FUNCTION_BLOCK "HF3_IMCC_DT_FB2711"	// FB 2711
VERSION : 0.1
VAR
  PT_DT : TIME  := T#45S;
  K4_DTS_A1 : FB 2712;
  K4_DTS_A2 : FB 2712;
  K4_DTS_A3 : FB 2712;
  DTS_A1 : FB 2712;
  DTS_A2 : FB 2712;
  DTS_A4 : FB 2712;
  DTS_A6 : FB 2712;
  UOF_DT_A1 : FB 2712;
  UOF_DT_A2 : FB 2712;
  UOF_DT_A3 : FB 2712;
  UOF_DT_A4 : FB 2712;
  DTS_A5 : FB 2712;
  DTS_A3 : FB 2712;
END_VAR
BEGIN
NETWORK
TITLE =  K4-DTS-A1
      A     "IMCC_LOCK".K4_XK_A1_Stop;
      =     L 0.0;
      BLD   103;
      BLD   14;
      =     L 7.0;
      L     DINO;
      T     LW 5;
      CDB;
      OPN   DI [LW 5];
      TAR2  LD 1;
      OPN   DI 2291;
      L     DIW 604;
      OPN   DI [LW 5];
      T     #K4_DTS_A1.IN_RD;
      OPN   DI 6040;
      L     DIW 152;
      OPN   DI [LW 5];
      T     #K4_DTS_A1.SCtrl;
      OPN   DI 7005;
      L     DIW 312;
      OPN   DI [LW 5];
      T     #K4_DTS_A1.H_P_ALL_Ctrl;
      A     L 0.0;
      =     #K4_DTS_A1.Stop;
      BLD   11;
      L     W#16#1002;
      T     LW 10;
      L     2;
      T     LW 12;
      L     7004;
      T     LW 14;
      L     P#DBX 58.0;
      T     LD 16;
      L     W#16#1002;
      T     LW 20;
      L     2;
      T     LW 22;
      L     DINO;
      T     LW 24;
      +AR2  P#12.0;
      TAR2;
      LAR2  LD 1;
      T     LD 26;
      UC    "BLKMOV";
      {     P#L 10.0, P#L 8.0, P#L 20.0 };
      BLD   11;
      L     W#16#1002;
      T     LW 10;
      L     2;
      T     LW 12;
      L     7005;
      T     LW 14;
      L     P#DBX 4.0;
      T     LD 16;
      L     W#16#1002;
      T     LW 20;
      L     2;
      T     LW 22;
      L     DINO;
      T     LW 24;
      +AR2  P#14.0;
      TAR2;
      LAR2  LD 1;
      T     LD 26;
      UC    "BLKMOV";
      {     P#L 10.0, P#L 8.0, P#L 20.0 };
      BLD   11;
      L     W#16#1002;
      T     LW 10;
      L     2;
      T     LW 12;
      L     7005;
      T     LW 14;
      L     P#DBX 34.0;
      T     LD 16;
      L     W#16#1002;
      T     LW 20;
      L     2;
      T     LW 22;
      L     DINO;
      T     LW 24;
      +AR2  P#16.0;
      TAR2;
      LAR2  LD 1;
      T     LD 26;
      UC    "BLKMOV";
      {     P#L 10.0, P#L 8.0, P#L 20.0 };
      L     DBD [AR2,P#0.0];
      T     #K4_DTS_A1.PT;
      +AR2  P#4.0;
      UC    "HF3_IMCC_DT_FB2712";
      LAR2  LD 1;
      L     #K4_DTS_A1.qnWR;
      OPN   DI 2292;
      T     DIW 124;
      OPN   DI [LW 5];
      L     #K4_DTS_A1.TOHMI;
      OPN   DI 6004;
      T     DIW 482;
      OPN   DI [LW 5];
      A     #K4_DTS_A1.Refuse;
      OPN   DI 7006;
      =     DIX 5.0;
      OPN   DI [LW 5];
      A     #K4_DTS_A1.Open;
      OPN   DI 2555;
      =     DIX 3.1;
      OPN   DI [LW 5];
      CDB;
      BLD   15;
      NOP   0;
NETWORK
TITLE =  K4-DTS-A2
      A     "IMCC_LOCK".K4_DT_A2_Open;
      =     L 0.0;
      BLD   103;
      BLD   14;
      =     L 7.0;
      L     DINO;
      T     LW 5;
      CDB;
      OPN   DI [LW 5];
      TAR2  LD 1;
      OPN   DI 2291;
      L     DIW 606;
      OPN   DI [LW 5];
      T     DIW [AR2,P#110.0];
      OPN   DI 6040;
      L     DIW 154;
      OPN   DI [LW 5];
      T     DIW [AR2,P#112.0];
      OPN   DI 7005;
      L     DIW 312;
      OPN   DI [LW 5];
      T     DIW [AR2,P#114.0];
      A     L 0.0;
      =     DIX [AR2,P#116.0];
      BLD   11;
      L     W#16#1002;
      T     LW 10;
      L     2;
      T     LW 12;
      L     7004;
      T     LW 14;
      L     P#DBX 60.0;
      T     LD 16;
      L     W#16#1002;
      T     LW 20;
      L     2;
      T     LW 22;
      L     DINO;
      T     LW 24;
      +AR2  P#118.0;
      TAR2;
      LAR2  LD 1;
      T     LD 26;
      UC    "BLKMOV";
      {     P#L 10.0, P#L 8.0, P#L 20.0 };
      BLD   11;
      L     W#16#1002;
      T     LW 10;
      L     2;
      T     LW 12;
      L     7005;
      T     LW 14;
      L     P#DBX 4.0;
      T     LD 16;
      L     W#16#1002;
      T     LW 20;
      L     2;
      T     LW 22;
      L     DINO;
      T     LW 24;
      +AR2  P#120.0;
      TAR2;
      LAR2  LD 1;
      T     LD 26;
      UC    "BLKMOV";
      {     P#L 10.0, P#L 8.0, P#L 20.0 };
      BLD   11;
      L     W#16#1002;
      T     LW 10;
      L     2;
      T     LW 12;
      L     7005;
      T     LW 14;
      L     P#DBX 34.0;
      T     LD 16;
      L     W#16#1002;
      T     LW 20;
      L     2;
      T     LW 22;
      L     DINO;
      T     LW 24;
      +AR2  P#122.0;
      TAR2;
      LAR2  LD 1;
      T     LD 26;
      UC    "BLKMOV";
      {     P#L 10.0, P#L 8.0, P#L 20.0 };
      L     DBD [AR2,P#0.0];
      T     DID [AR2,P#124.0];
      +AR2  P#110.0;
      UC    "HF3_IMCC_DT_FB2712";
      LAR2  LD 1;
      L     DIW [AR2,P#128.0];
      OPN   DI 2292;
      T     DIW 126;
      OPN   DI [LW 5];
      L     DIW [AR2,P#130.0];
      OPN   DI 6004;
      T     DIW 484;
      OPN   DI [LW 5];
      A     DIX [AR2,P#132.0];
      OPN   DI 7006;
      =     DIX 5.1;
      OPN   DI [LW 5];
      A     DIX [AR2,P#132.1];
      OPN   DI 2555;
      =     DIX 3.2;
      OPN   DI [LW 5];
      CDB;
      BLD   15;
      NOP   0;
NETWORK
TITLE =  K4-DTS-A3
      A(;
      O     "IMCC_LOCK".K4_HPF_A1_Stop;
      O     "IMCC_LOCK".K4_XK_A1_Stop;
      );
      =     L 0.0;
      BLD   103;
      BLD   14;
      =     L 7.0;
      L     DINO;
      T     LW 5;
      CDB;
      OPN   DI [LW 5];
      TAR2  LD 1;
      OPN   DI 2291;
      L     DIW 608;
      OPN   DI [LW 5];
      T     DIW [AR2,P#216.0];
      OPN   DI 6040;
      L     DIW 156;
      OPN   DI [LW 5];
      T     DIW [AR2,P#218.0];
      OPN   DI 7005;
      L     DIW 312;
      OPN   DI [LW 5];
      T     DIW [AR2,P#220.0];
      A     L 0.0;
      =     DIX [AR2,P#222.0];
      BLD   11;
      L     W#16#1002;
      T     LW 10;
      L     2;
      T     LW 12;
      L     7004;
      T     LW 14;
      L     P#DBX 62.0;
      T     LD 16;
      L     W#16#1002;
      T     LW 20;
      L     2;
      T     LW 22;
      L     DINO;
      T     LW 24;
      +AR2  P#224.0;
      TAR2;
      LAR2  LD 1;
      T     LD 26;
      UC    "BLKMOV";
      {     P#L 10.0, P#L 8.0, P#L 20.0 };
      BLD   11;
      L     W#16#1002;
      T     LW 10;
      L     2;
      T     LW 12;
      L     7005;
      T     LW 14;
      L     P#DBX 4.0;
      T     LD 16;
      L     W#16#1002;
      T     LW 20;
      L     2;
      T     LW 22;
      L     DINO;
      T     LW 24;
      +AR2  P#226.0;
      TAR2;
      LAR2  LD 1;
      T     LD 26;
      UC    "BLKMOV";
      {     P#L 10.0, P#L 8.0, P#L 20.0 };
      BLD   11;
      L     W#16#1002;
      T     LW 10;
      L     2;
      T     LW 12;
      L     7005;
      T     LW 14;
      L     P#DBX 34.0;
      T     LD 16;
      L     W#16#1002;
      T     LW 20;
      L     2;
      T     LW 22;
      L     DINO;
      T     LW 24;
      +AR2  P#228.0;
      TAR2;
      LAR2  LD 1;
      T     LD 26;
      UC    "BLKMOV";
      {     P#L 10.0, P#L 8.0, P#L 20.0 };
      L     DBD [AR2,P#0.0];
      T     DID [AR2,P#230.0];
      +AR2  P#216.0;
      UC    "HF3_IMCC_DT_FB2712";
      LAR2  LD 1;
      L     DIW [AR2,P#234.0];
      OPN   DI 2292;
      T     DIW 128;
      OPN   DI [LW 5];
      L     DIW [AR2,P#236.0];
      OPN   DI 6004;
      T     DIW 486;
      OPN   DI [LW 5];
      A     DIX [AR2,P#238.0];
      OPN   DI 7006;
      =     DIX 5.2;
      OPN   DI [LW 5];
      A     DIX [AR2,P#238.1];
      OPN   DI 2555;
      =     DIX 3.3;
      OPN   DI [LW 5];
      CDB;
      BLD   15;
      NOP   0;
NETWORK
TITLE = DTS-A1
      A     "Always1";
      =     L 0.0;
      BLD   103;
      BLD   14;
      =     L 7.0;
      L     DINO;
      T     LW 5;
      CDB;
      OPN   DI [LW 5];
      TAR2  LD 1;
      OPN   DI 2291;
      L     DIW 676;
      OPN   DI [LW 5];
      T     DIW [AR2,P#322.0];
      OPN   DI 6040;
      L     DIW 60;
      OPN   DI [LW 5];
      T     DIW [AR2,P#324.0];
      OPN   DI 7005;
      L     DIW 312;
      OPN   DI [LW 5];
      T     DIW [AR2,P#326.0];
      A     L 0.0;
      =     DIX [AR2,P#328.0];
      BLD   11;
      L     W#16#1002;
      T     LW 10;
      L     2;
      T     LW 12;
      L     7004;
      T     LW 14;
      L     P#DBX 4.0;
      T     LD 16;
      L     W#16#1002;
      T     LW 20;
      L     2;
      T     LW 22;
      L     DINO;
      T     LW 24;
      +AR2  P#330.0;
      TAR2;
      LAR2  LD 1;
      T     LD 26;
      UC    "BLKMOV";
      {     P#L 10.0, P#L 8.0, P#L 20.0 };
      BLD   11;
      L     W#16#1002;
      T     LW 10;
      L     2;
      T     LW 12;
      L     7005;
      T     LW 14;
      L     P#DBX 0.0;
      T     LD 16;
      L     W#16#1002;
      T     LW 20;
      L     2;
      T     LW 22;
      L     DINO;
      T     LW 24;
      +AR2  P#332.0;
      TAR2;
      LAR2  LD 1;
      T     LD 26;
      UC    "BLKMOV";
      {     P#L 10.0, P#L 8.0, P#L 20.0 };
      BLD   11;
      L     W#16#1002;
      T     LW 10;
      L     2;
      T     LW 12;
      L     7005;
      T     LW 14;
      L     P#DBX 30.0;
      T     LD 16;
      L     W#16#1002;
      T     LW 20;
      L     2;
      T     LW 22;
      L     DINO;
      T     LW 24;
      +AR2  P#334.0;
      TAR2;
      LAR2  LD 1;
      T     LD 26;
      UC    "BLKMOV";
      {     P#L 10.0, P#L 8.0, P#L 20.0 };
      L     DBD [AR2,P#0.0];
      T     DID [AR2,P#336.0];
      +AR2  P#322.0;
      UC    "HF3_IMCC_DT_FB2712";
      LAR2  LD 1;
      L     DIW [AR2,P#340.0];
      OPN   DI 2292;
      T     DIW 196;
      OPN   DI [LW 5];
      L     DIW [AR2,P#342.0];
      OPN   DI 6004;
      T     DIW 518;
      OPN   DI [LW 5];
      A     DIX [AR2,P#344.0];
      OPN   DI 7006;
      =     DIX 2.0;
      OPN   DI [LW 5];
      A     DIX [AR2,P#344.1];
      OPN   DI 2555;
      =     DIX 0.2;
      OPN   DI [LW 5];
      CDB;
      BLD   15;
      NOP   0;
NETWORK
TITLE = DTS-A2
      A     "Always1";
      =     L 0.0;
      BLD   103;
      BLD   14;
      =     L 7.0;
      L     DINO;
      T     LW 5;
      CDB;
      OPN   DI [LW 5];
      TAR2  LD 1;
      OPN   DI 2291;
      L     DIW 678;
      OPN   DI [LW 5];
      T     DIW [AR2,P#428.0];
      OPN   DI 6040;
      L     DIW 62;
      OPN   DI [LW 5];
      T     DIW [AR2,P#430.0];
      OPN   DI 7005;
      L     DIW 312;
      OPN   DI [LW 5];
      T     DIW [AR2,P#432.0];
      A     L 0.0;
      =     DIX [AR2,P#434.0];
      BLD   11;
      L     W#16#1002;
      T     LW 10;
      L     2;
      T     LW 12;
      L     7004;
      T     LW 14;
      L     P#DBX 6.0;
      T     LD 16;
      L     W#16#1002;
      T     LW 20;
      L     2;
      T     LW 22;
      L     DINO;
      T     LW 24;
      +AR2  P#436.0;
      TAR2;
      LAR2  LD 1;
      T     LD 26;
      UC    "BLKMOV";
      {     P#L 10.0, P#L 8.0, P#L 20.0 };
      BLD   11;
      L     W#16#1002;
      T     LW 10;
      L     2;
      T     LW 12;
      L     7005;
      T     LW 14;
      L     P#DBX 0.0;
      T     LD 16;
      L     W#16#1002;
      T     LW 20;
      L     2;
      T     LW 22;
      L     DINO;
      T     LW 24;
      +AR2  P#438.0;
      TAR2;
      LAR2  LD 1;
      T     LD 26;
      UC    "BLKMOV";
      {     P#L 10.0, P#L 8.0, P#L 20.0 };
      BLD   11;
      L     W#16#1002;
      T     LW 10;
      L     2;
      T     LW 12;
      L     7005;
      T     LW 14;
      L     P#DBX 30.0;
      T     LD 16;
      L     W#16#1002;
      T     LW 20;
      L     2;
      T     LW 22;
      L     DINO;
      T     LW 24;
      +AR2  P#440.0;
      TAR2;
      LAR2  LD 1;
      T     LD 26;
      UC    "BLKMOV";
      {     P#L 10.0, P#L 8.0, P#L 20.0 };
      L     DBD [AR2,P#0.0];
      T     DID [AR2,P#442.0];
      +AR2  P#428.0;
      UC    "HF3_IMCC_DT_FB2712";
      LAR2  LD 1;
      L     DIW [AR2,P#446.0];
      OPN   DI 2292;
      T     DIW 198;
      OPN   DI [LW 5];
      L     DIW [AR2,P#448.0];
      OPN   DI 6004;
      T     DIW 520;
      OPN   DI [LW 5];
      A     DIX [AR2,P#450.0];
      OPN   DI 7006;
      =     DIX 2.1;
      OPN   DI [LW 5];
      A     DIX [AR2,P#450.1];
      OPN   DI 2555;
      =     DIX 0.3;
      OPN   DI [LW 5];
      CDB;
      BLD   15;
      NOP   0;
NETWORK
TITLE = DTS-A3
      A     "Always1";
      =     L 0.0;
      BLD   103;
      BLD   14;
      =     L 7.0;
      L     DINO;
      T     LW 5;
      CDB;
      OPN   DI [LW 5];
      TAR2  LD 1;
      OPN   DI 2291;
      L     DIW 680;
      OPN   DI [LW 5];
      T     DIW [AR2,P#1276.0];
      OPN   DI 6040;
      L     DIW 64;
      OPN   DI [LW 5];
      T     DIW [AR2,P#1278.0];
      OPN   DI 7005;
      L     DIW 312;
      OPN   DI [LW 5];
      T     DIW [AR2,P#1280.0];
      A     L 0.0;
      =     DIX [AR2,P#1282.0];
      BLD   11;
      L     W#16#1002;
      T     LW 10;
      L     2;
      T     LW 12;
      L     7004;
      T     LW 14;
      L     P#DBX 8.0;
      T     LD 16;
      L     W#16#1002;
      T     LW 20;
      L     2;
      T     LW 22;
      L     DINO;
      T     LW 24;
      +AR2  P#1284.0;
      TAR2;
      LAR2  LD 1;
      T     LD 26;
      UC    "BLKMOV";
      {     P#L 10.0, P#L 8.0, P#L 20.0 };
      BLD   11;
      L     W#16#1002;
      T     LW 10;
      L     2;
      T     LW 12;
      L     7005;
      T     LW 14;
      L     P#DBX 0.0;
      T     LD 16;
      L     W#16#1002;
      T     LW 20;
      L     2;
      T     LW 22;
      L     DINO;
      T     LW 24;
      +AR2  P#1286.0;
      TAR2;
      LAR2  LD 1;
      T     LD 26;
      UC    "BLKMOV";
      {     P#L 10.0, P#L 8.0, P#L 20.0 };
      BLD   11;
      L     W#16#1002;
      T     LW 10;
      L     2;
      T     LW 12;
      L     7005;
      T     LW 14;
      L     P#DBX 30.0;
      T     LD 16;
      L     W#16#1002;
      T     LW 20;
      L     2;
      T     LW 22;
      L     DINO;
      T     LW 24;
      +AR2  P#1288.0;
      TAR2;
      LAR2  LD 1;
      T     LD 26;
      UC    "BLKMOV";
      {     P#L 10.0, P#L 8.0, P#L 20.0 };
      L     DBD [AR2,P#0.0];
      T     DID [AR2,P#1290.0];
      +AR2  P#1276.0;
      UC    "HF3_IMCC_DT_FB2712";
      LAR2  LD 1;
      L     DIW [AR2,P#1294.0];
      OPN   DI 2292;
      T     DIW 200;
      OPN   DI [LW 5];
      L     DIW [AR2,P#1296.0];
      OPN   DI 6004;
      T     DIW 522;
      OPN   DI [LW 5];
      A     DIX [AR2,P#1298.0];
      OPN   DI 7006;
      =     DIX 2.2;
      OPN   DI [LW 5];
      A     DIX [AR2,P#1298.1];
      OPN   DI 2555;
      =     DIX 0.4;
      OPN   DI [LW 5];
      CDB;
      BLD   15;
      NOP   0;
NETWORK
TITLE = DTS-A4
      A     "Always1";
      =     L 0.0;
      BLD   103;
      BLD   14;
      =     L 7.0;
      L     DINO;
      T     LW 5;
      CDB;
      OPN   DI [LW 5];
      TAR2  LD 1;
      OPN   DI 2291;
      L     DIW 682;
      OPN   DI [LW 5];
      T     DIW [AR2,P#534.0];
      OPN   DI 6040;
      L     DIW 66;
      OPN   DI [LW 5];
      T     DIW [AR2,P#536.0];
      OPN   DI 7005;
      L     DIW 312;
      OPN   DI [LW 5];
      T     DIW [AR2,P#538.0];
      A     L 0.0;
      =     DIX [AR2,P#540.0];
      BLD   11;
      L     W#16#1002;
      T     LW 10;
      L     2;
      T     LW 12;
      L     7004;
      T     LW 14;
      L     P#DBX 10.0;
      T     LD 16;
      L     W#16#1002;
      T     LW 20;
      L     2;
      T     LW 22;
      L     DINO;
      T     LW 24;
      +AR2  P#542.0;
      TAR2;
      LAR2  LD 1;
      T     LD 26;
      UC    "BLKMOV";
      {     P#L 10.0, P#L 8.0, P#L 20.0 };
      BLD   11;
      L     W#16#1002;
      T     LW 10;
      L     2;
      T     LW 12;
      L     7005;
      T     LW 14;
      L     P#DBX 0.0;
      T     LD 16;
      L     W#16#1002;
      T     LW 20;
      L     2;
      T     LW 22;
      L     DINO;
      T     LW 24;
      +AR2  P#544.0;
      TAR2;
      LAR2  LD 1;
      T     LD 26;
      UC    "BLKMOV";
      {     P#L 10.0, P#L 8.0, P#L 20.0 };
      BLD   11;
      L     W#16#1002;
      T     LW 10;
      L     2;
      T     LW 12;
      L     7005;
      T     LW 14;
      L     P#DBX 30.0;
      T     LD 16;
      L     W#16#1002;
      T     LW 20;
      L     2;
      T     LW 22;
      L     DINO;
      T     LW 24;
      +AR2  P#546.0;
      TAR2;
      LAR2  LD 1;
      T     LD 26;
      UC    "BLKMOV";
      {     P#L 10.0, P#L 8.0, P#L 20.0 };
      L     DBD [AR2,P#0.0];
      T     DID [AR2,P#548.0];
      +AR2  P#534.0;
      UC    "HF3_IMCC_DT_FB2712";
      LAR2  LD 1;
      L     DIW [AR2,P#552.0];
      OPN   DI 2292;
      T     DIW 202;
      OPN   DI [LW 5];
      L     DIW [AR2,P#554.0];
      OPN   DI 6004;
      T     DIW 524;
      OPN   DI [LW 5];
      A     DIX [AR2,P#556.0];
      OPN   DI 7006;
      =     DIX 2.3;
      OPN   DI [LW 5];
      A     DIX [AR2,P#556.1];
      OPN   DI 2555;
      =     DIX 0.5;
      OPN   DI [LW 5];
      CDB;
      BLD   15;
      NOP   0;
NETWORK
TITLE = DTS-A5
      A     "Always1";
      =     L 0.0;
      BLD   103;
      BLD   14;
      =     L 7.0;
      L     DINO;
      T     LW 5;
      CDB;
      OPN   DI [LW 5];
      TAR2  LD 1;
      OPN   DI 2291;
      L     DIW 684;
      OPN   DI [LW 5];
      T     DIW [AR2,P#1170.0];
      OPN   DI 6040;
      L     DIW 68;
      OPN   DI [LW 5];
      T     DIW [AR2,P#1172.0];
      OPN   DI 7005;
      L     DIW 312;
      OPN   DI [LW 5];
      T     DIW [AR2,P#1174.0];
      A     L 0.0;
      =     DIX [AR2,P#1176.0];
      BLD   11;
      L     W#16#1002;
      T     LW 10;
      L     2;
      T     LW 12;
      L     7004;
      T     LW 14;
      L     P#DBX 12.0;
      T     LD 16;
      L     W#16#1002;
      T     LW 20;
      L     2;
      T     LW 22;
      L     DINO;
      T     LW 24;
      +AR2  P#1178.0;
      TAR2;
      LAR2  LD 1;
      T     LD 26;
      UC    "BLKMOV";
      {     P#L 10.0, P#L 8.0, P#L 20.0 };
      BLD   11;
      L     W#16#1002;
      T     LW 10;
      L     2;
      T     LW 12;
      L     7005;
      T     LW 14;
      L     P#DBX 0.0;
      T     LD 16;
      L     W#16#1002;
      T     LW 20;
      L     2;
      T     LW 22;
      L     DINO;
      T     LW 24;
      +AR2  P#1180.0;
      TAR2;
      LAR2  LD 1;
      T     LD 26;
      UC    "BLKMOV";
      {     P#L 10.0, P#L 8.0, P#L 20.0 };
      BLD   11;
      L     W#16#1002;
      T     LW 10;
      L     2;
      T     LW 12;
      L     7005;
      T     LW 14;
      L     P#DBX 30.0;
      T     LD 16;
      L     W#16#1002;
      T     LW 20;
      L     2;
      T     LW 22;
      L     DINO;
      T     LW 24;
      +AR2  P#1182.0;
      TAR2;
      LAR2  LD 1;
      T     LD 26;
      UC    "BLKMOV";
      {     P#L 10.0, P#L 8.0, P#L 20.0 };
      L     DBD [AR2,P#0.0];
      T     DID [AR2,P#1184.0];
      +AR2  P#1170.0;
      UC    "HF3_IMCC_DT_FB2712";
      LAR2  LD 1;
      L     DIW [AR2,P#1188.0];
      OPN   DI 2292;
      T     DIW 204;
      OPN   DI [LW 5];
      L     DIW [AR2,P#1190.0];
      OPN   DI 6004;
      T     DIW 526;
      OPN   DI [LW 5];
      A     DIX [AR2,P#1192.0];
      OPN   DI 7006;
      =     DIX 2.4;
      OPN   DI [LW 5];
      A     DIX [AR2,P#1192.1];
      OPN   DI 2555;
      =     DIX 0.6;
      OPN   DI [LW 5];
      CDB;
      BLD   15;
      NOP   0;
NETWORK
TITLE = DTS-A6
      A     "Always1";
      =     L 0.0;
      BLD   103;
      BLD   14;
      =     L 7.0;
      L     DINO;
      T     LW 5;
      CDB;
      OPN   DI [LW 5];
      TAR2  LD 1;
      OPN   DI 2291;
      L     DIW 686;
      OPN   DI [LW 5];
      T     DIW [AR2,P#640.0];
      OPN   DI 6040;
      L     DIW 70;
      OPN   DI [LW 5];
      T     DIW [AR2,P#642.0];
      OPN   DI 7005;
      L     DIW 312;
      OPN   DI [LW 5];
      T     DIW [AR2,P#644.0];
      A     L 0.0;
      =     DIX [AR2,P#646.0];
      BLD   11;
      L     W#16#1002;
      T     LW 10;
      L     2;
      T     LW 12;
      L     7004;
      T     LW 14;
      L     P#DBX 14.0;
      T     LD 16;
      L     W#16#1002;
      T     LW 20;
      L     2;
      T     LW 22;
      L     DINO;
      T     LW 24;
      +AR2  P#648.0;
      TAR2;
      LAR2  LD 1;
      T     LD 26;
      UC    "BLKMOV";
      {     P#L 10.0, P#L 8.0, P#L 20.0 };
      BLD   11;
      L     W#16#1002;
      T     LW 10;
      L     2;
      T     LW 12;
      L     7005;
      T     LW 14;
      L     P#DBX 0.0;
      T     LD 16;
      L     W#16#1002;
      T     LW 20;
      L     2;
      T     LW 22;
      L     DINO;
      T     LW 24;
      +AR2  P#650.0;
      TAR2;
      LAR2  LD 1;
      T     LD 26;
      UC    "BLKMOV";
      {     P#L 10.0, P#L 8.0, P#L 20.0 };
      BLD   11;
      L     W#16#1002;
      T     LW 10;
      L     2;
      T     LW 12;
      L     7005;
      T     LW 14;
      L     P#DBX 30.0;
      T     LD 16;
      L     W#16#1002;
      T     LW 20;
      L     2;
      T     LW 22;
      L     DINO;
      T     LW 24;
      +AR2  P#652.0;
      TAR2;
      LAR2  LD 1;
      T     LD 26;
      UC    "BLKMOV";
      {     P#L 10.0, P#L 8.0, P#L 20.0 };
      L     DBD [AR2,P#0.0];
      T     DID [AR2,P#654.0];
      +AR2  P#640.0;
      UC    "HF3_IMCC_DT_FB2712";
      LAR2  LD 1;
      L     DIW [AR2,P#658.0];
      OPN   DI 2292;
      T     DIW 206;
      OPN   DI [LW 5];
      L     DIW [AR2,P#660.0];
      OPN   DI 6004;
      T     DIW 528;
      OPN   DI [LW 5];
      A     DIX [AR2,P#662.0];
      OPN   DI 7006;
      =     DIX 2.5;
      OPN   DI [LW 5];
      A     DIX [AR2,P#662.1];
      OPN   DI 2555;
      =     DIX 0.7;
      OPN   DI [LW 5];
      CDB;
      BLD   15;
      NOP   0;
NETWORK
TITLE = UOF_DTS_A1
      A     "Always1";
      =     L 0.0;
      BLD   103;
      BLD   14;
      =     L 7.0;
      L     DINO;
      T     LW 5;
      CDB;
      OPN   DI [LW 5];
      TAR2  LD 1;
      OPN   DI 2291;
      L     DIW 668;
      OPN   DI [LW 5];
      T     DIW [AR2,P#746.0];
      OPN   DI 6040;
      L     DIW 106;
      OPN   DI [LW 5];
      T     DIW [AR2,P#748.0];
      OPN   DI 7005;
      L     DIW 312;
      OPN   DI [LW 5];
      T     DIW [AR2,P#750.0];
      A     L 0.0;
      =     DIX [AR2,P#752.0];
      BLD   11;
      L     W#16#1002;
      T     LW 10;
      L     2;
      T     LW 12;
      L     7004;
      T     LW 14;
      L     P#DBX 38.0;
      T     LD 16;
      L     W#16#1002;
      T     LW 20;
      L     2;
      T     LW 22;
      L     DINO;
      T     LW 24;
      +AR2  P#754.0;
      TAR2;
      LAR2  LD 1;
      T     LD 26;
      UC    "BLKMOV";
      {     P#L 10.0, P#L 8.0, P#L 20.0 };
      BLD   11;
      L     W#16#1002;
      T     LW 10;
      L     2;
      T     LW 12;
      L     7005;
      T     LW 14;
      L     P#DBX 0.0;
      T     LD 16;
      L     W#16#1002;
      T     LW 20;
      L     2;
      T     LW 22;
      L     DINO;
      T     LW 24;
      +AR2  P#756.0;
      TAR2;
      LAR2  LD 1;
      T     LD 26;
      UC    "BLKMOV";
      {     P#L 10.0, P#L 8.0, P#L 20.0 };
      BLD   11;
      L     W#16#1002;
      T     LW 10;
      L     2;
      T     LW 12;
      L     7005;
      T     LW 14;
      L     P#DBX 30.0;
      T     LD 16;
      L     W#16#1002;
      T     LW 20;
      L     2;
      T     LW 22;
      L     DINO;
      T     LW 24;
      +AR2  P#758.0;
      TAR2;
      LAR2  LD 1;
      T     LD 26;
      UC    "BLKMOV";
      {     P#L 10.0, P#L 8.0, P#L 20.0 };
      L     DBD [AR2,P#0.0];
      T     DID [AR2,P#760.0];
      +AR2  P#746.0;
      UC    "HF3_IMCC_DT_FB2712";
      LAR2  LD 1;
      L     DIW [AR2,P#764.0];
      OPN   DI 2292;
      T     DIW 188;
      OPN   DI [LW 5];
      L     DIW [AR2,P#766.0];
      OPN   DI 6004;
      T     DIW 510;
      OPN   DI [LW 5];
      A     DIX [AR2,P#768.0];
      OPN   DI 7006;
      =     DIX 4.2;
      OPN   DI [LW 5];
      CDB;
      BLD   15;
      NOP   0;
NETWORK
TITLE = UOF_DTS_A2
      A     "Always1";
      =     L 0.0;
      BLD   103;
      BLD   14;
      =     L 7.0;
      L     DINO;
      T     LW 5;
      CDB;
      OPN   DI [LW 5];
      TAR2  LD 1;
      OPN   DI 2291;
      L     DIW 670;
      OPN   DI [LW 5];
      T     DIW [AR2,P#852.0];
      OPN   DI 6040;
      L     DIW 108;
      OPN   DI [LW 5];
      T     DIW [AR2,P#854.0];
      OPN   DI 7005;
      L     DIW 312;
      OPN   DI [LW 5];
      T     DIW [AR2,P#856.0];
      A     L 0.0;
      =     DIX [AR2,P#858.0];
      BLD   11;
      L     W#16#1002;
      T     LW 10;
      L     2;
      T     LW 12;
      L     7004;
      T     LW 14;
      L     P#DBX 40.0;
      T     LD 16;
      L     W#16#1002;
      T     LW 20;
      L     2;
      T     LW 22;
      L     DINO;
      T     LW 24;
      +AR2  P#860.0;
      TAR2;
      LAR2  LD 1;
      T     LD 26;
      UC    "BLKMOV";
      {     P#L 10.0, P#L 8.0, P#L 20.0 };
      BLD   11;
      L     W#16#1002;
      T     LW 10;
      L     2;
      T     LW 12;
      L     7005;
      T     LW 14;
      L     P#DBX 0.0;
      T     LD 16;
      L     W#16#1002;
      T     LW 20;
      L     2;
      T     LW 22;
      L     DINO;
      T     LW 24;
      +AR2  P#862.0;
      TAR2;
      LAR2  LD 1;
      T     LD 26;
      UC    "BLKMOV";
      {     P#L 10.0, P#L 8.0, P#L 20.0 };
      BLD   11;
      L     W#16#1002;
      T     LW 10;
      L     2;
      T     LW 12;
      L     7005;
      T     LW 14;
      L     P#DBX 30.0;
      T     LD 16;
      L     W#16#1002;
      T     LW 20;
      L     2;
      T     LW 22;
      L     DINO;
      T     LW 24;
      +AR2  P#864.0;
      TAR2;
      LAR2  LD 1;
      T     LD 26;
      UC    "BLKMOV";
      {     P#L 10.0, P#L 8.0, P#L 20.0 };
      L     DBD [AR2,P#0.0];
      T     DID [AR2,P#866.0];
      +AR2  P#852.0;
      UC    "HF3_IMCC_DT_FB2712";
      LAR2  LD 1;
      L     DIW [AR2,P#870.0];
      OPN   DI 2292;
      T     DIW 190;
      OPN   DI [LW 5];
      L     DIW [AR2,P#872.0];
      OPN   DI 6004;
      T     DIW 512;
      OPN   DI [LW 5];
      A     DIX [AR2,P#874.0];
      OPN   DI 7006;
      =     DIX 4.3;
      OPN   DI [LW 5];
      CDB;
      BLD   15;
      NOP   0;
NETWORK
TITLE = UOF_DTS_A3
      A     "Always1";
      =     L 0.0;
      BLD   103;
      BLD   14;
      =     L 7.0;
      L     DINO;
      T     LW 5;
      CDB;
      OPN   DI [LW 5];
      TAR2  LD 1;
      OPN   DI 2291;
      L     DIW 672;
      OPN   DI [LW 5];
      T     DIW [AR2,P#958.0];
      OPN   DI 6040;
      L     DIW 110;
      OPN   DI [LW 5];
      T     DIW [AR2,P#960.0];
      OPN   DI 7005;
      L     DIW 312;
      OPN   DI [LW 5];
      T     DIW [AR2,P#962.0];
      A     L 0.0;
      =     DIX [AR2,P#964.0];
      BLD   11;
      L     W#16#1002;
      T     LW 10;
      L     2;
      T     LW 12;
      L     7004;
      T     LW 14;
      L     P#DBX 42.0;
      T     LD 16;
      L     W#16#1002;
      T     LW 20;
      L     2;
      T     LW 22;
      L     DINO;
      T     LW 24;
      +AR2  P#966.0;
      TAR2;
      LAR2  LD 1;
      T     LD 26;
      UC    "BLKMOV";
      {     P#L 10.0, P#L 8.0, P#L 20.0 };
      BLD   11;
      L     W#16#1002;
      T     LW 10;
      L     2;
      T     LW 12;
      L     7005;
      T     LW 14;
      L     P#DBX 0.0;
      T     LD 16;
      L     W#16#1002;
      T     LW 20;
      L     2;
      T     LW 22;
      L     DINO;
      T     LW 24;
      +AR2  P#968.0;
      TAR2;
      LAR2  LD 1;
      T     LD 26;
      UC    "BLKMOV";
      {     P#L 10.0, P#L 8.0, P#L 20.0 };
      BLD   11;
      L     W#16#1002;
      T     LW 10;
      L     2;
      T     LW 12;
      L     7005;
      T     LW 14;
      L     P#DBX 30.0;
      T     LD 16;
      L     W#16#1002;
      T     LW 20;
      L     2;
      T     LW 22;
      L     DINO;
      T     LW 24;
      +AR2  P#970.0;
      TAR2;
      LAR2  LD 1;
      T     LD 26;
      UC    "BLKMOV";
      {     P#L 10.0, P#L 8.0, P#L 20.0 };
      L     DBD [AR2,P#0.0];
      T     DID [AR2,P#972.0];
      +AR2  P#958.0;
      UC    "HF3_IMCC_DT_FB2712";
      LAR2  LD 1;
      L     DIW [AR2,P#976.0];
      OPN   DI 2292;
      T     DIW 192;
      OPN   DI [LW 5];
      L     DIW [AR2,P#978.0];
      OPN   DI 6004;
      T     DIW 514;
      OPN   DI [LW 5];
      A     DIX [AR2,P#980.0];
      OPN   DI 7006;
      =     DIX 4.4;
      OPN   DI [LW 5];
      CDB;
      BLD   15;
      NOP   0;
NETWORK
TITLE = UOF_DTS_A4
      A     "Always1";
      =     L 0.0;
      BLD   103;
      BLD   14;
      =     L 7.0;
      L     DINO;
      T     LW 5;
      CDB;
      OPN   DI [LW 5];
      TAR2  LD 1;
      OPN   DI 2291;
      L     DIW 674;
      OPN   DI [LW 5];
      T     DIW [AR2,P#1064.0];
      OPN   DI 6040;
      L     DIW 112;
      OPN   DI [LW 5];
      T     DIW [AR2,P#1066.0];
      OPN   DI 7005;
      L     DIW 312;
      OPN   DI [LW 5];
      T     DIW [AR2,P#1068.0];
      A     L 0.0;
      =     DIX [AR2,P#1070.0];
      BLD   11;
      L     W#16#1002;
      T     LW 10;
      L     2;
      T     LW 12;
      L     7004;
      T     LW 14;
      L     P#DBX 44.0;
      T     LD 16;
      L     W#16#1002;
      T     LW 20;
      L     2;
      T     LW 22;
      L     DINO;
      T     LW 24;
      +AR2  P#1072.0;
      TAR2;
      LAR2  LD 1;
      T     LD 26;
      UC    "BLKMOV";
      {     P#L 10.0, P#L 8.0, P#L 20.0 };
      BLD   11;
      L     W#16#1002;
      T     LW 10;
      L     2;
      T     LW 12;
      L     7005;
      T     LW 14;
      L     P#DBX 0.0;
      T     LD 16;
      L     W#16#1002;
      T     LW 20;
      L     2;
      T     LW 22;
      L     DINO;
      T     LW 24;
      +AR2  P#1074.0;
      TAR2;
      LAR2  LD 1;
      T     LD 26;
      UC    "BLKMOV";
      {     P#L 10.0, P#L 8.0, P#L 20.0 };
      BLD   11;
      L     W#16#1002;
      T     LW 10;
      L     2;
      T     LW 12;
      L     7005;
      T     LW 14;
      L     P#DBX 30.0;
      T     LD 16;
      L     W#16#1002;
      T     LW 20;
      L     2;
      T     LW 22;
      L     DINO;
      T     LW 24;
      +AR2  P#1076.0;
      TAR2;
      LAR2  LD 1;
      T     LD 26;
      UC    "BLKMOV";
      {     P#L 10.0, P#L 8.0, P#L 20.0 };
      L     DBD [AR2,P#0.0];
      T     DID [AR2,P#1078.0];
      +AR2  P#1064.0;
      UC    "HF3_IMCC_DT_FB2712";
      LAR2  LD 1;
      L     DIW [AR2,P#1082.0];
      OPN   DI 2292;
      T     DIW 194;
      OPN   DI [LW 5];
      L     DIW [AR2,P#1084.0];
      OPN   DI 6004;
      T     DIW 516;
      OPN   DI [LW 5];
      A     DIX [AR2,P#1086.0];
      OPN   DI 7006;
      =     DIX 4.5;
      OPN   DI [LW 5];
      CDB;
      BLD   15;
      NOP   0;
END_FUNCTION_BLOCK

FUNCTION_BLOCK "HF3_IMCC_DT_FB2712"	// FB 2712
VERSION : 0.1
VAR_INPUT
  IN_RD : WORD ;
  SCtrl : WORD ;	//01-单控模块234-开半开关
  H_P_ALL_Ctrl : WORD ;	//全局命令
  Stop : BOOL ;	//连锁信号
  MCtrl : ARRAY  [0 .. 3 ] OF //0-开阀1-关阀
  BOOL ;
  Mode : ARRAY  [0 .. 15 ] OF //0-开始1-结束2-执行中
  BOOL ;
  ALL : ARRAY  [0 .. 15 ] OF //012-单控模控时间表
  BOOL ;
  PT : TIME ;	//设备动作超时
END_VAR
VAR_OUTPUT
  qnWR : WORD ;	//阀控制信息
  TOHMI : WORD ;
  Refuse : BOOL ;	//模式不符
  Open : BOOL ;	//阀控制信息
END_VAR
VAR
  qtwr_temp : WORD ;
  SCtrl_Temp : ARRAY  [0 .. 15 ] OF //01-单控模234-开半关
  BOOL ;
  DI_Temp : ARRAY  [0 .. 15 ] OF //234-开半开关
  BOOL ;
  DO_Temp : ARRAY  [0 .. 15 ] OF BOOL ;
  H_P_ALL_Ctrl_Temp : ARRAY  [0 .. 15 ] OF BOOL ;
  Ctrl : ARRAY  [0 .. 15 ] OF //012-开半开关
  BOOL ;
  Latch : ARRAY  [0 .. 15 ] OF //控制锁定
  BOOL ;
  SFlag : BOOL ;	//单控标志
  QTout : BOOL ;
  Timeout : BOOL ;	//设备动作超时
  McFlag : BOOL ;	//检修牌
  SingTout : BOOL ;
  FireAlarm : BOOL ;	//火灾信号
  BlockAlarm : BOOL ;	//阻塞信号
  TON1 : SFB 4;
  Ton2 : SFB 4;
  TON3 : SFB 4;
END_VAR
BEGIN
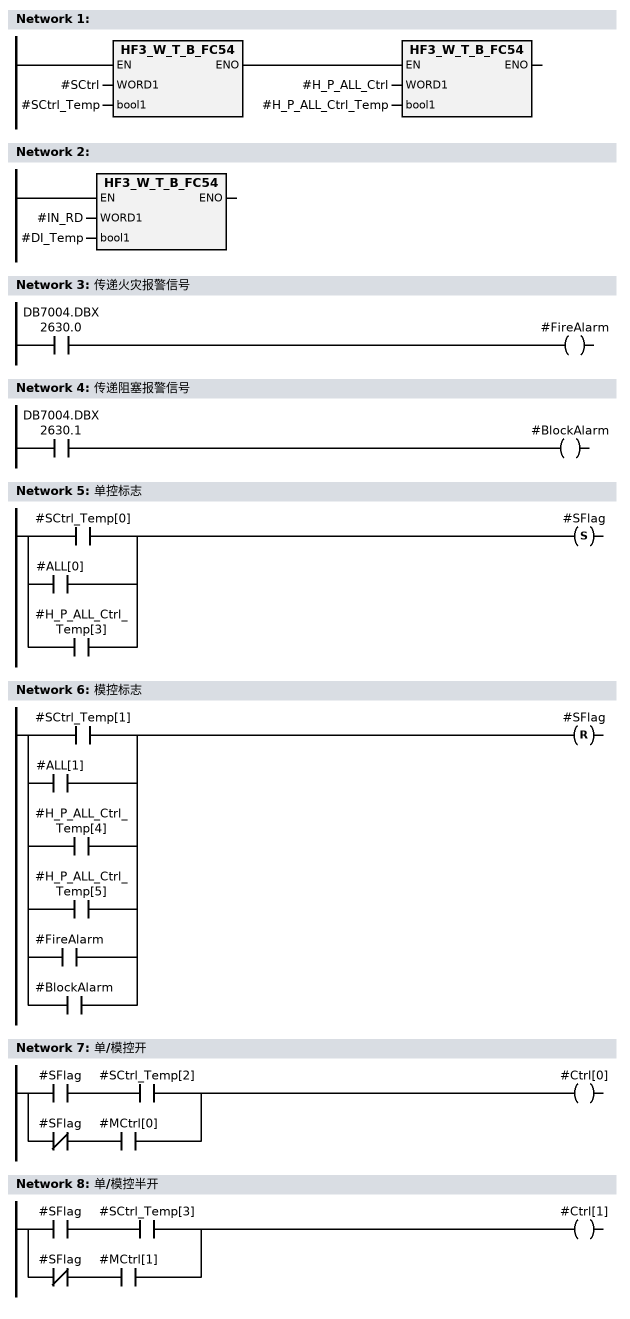
NETWORK
TITLE =
      A(;
      CALL  "HF3_W_T_B_FC54" (
           WORD1                    := #SCtrl,
           bool1                    := #SCtrl_Temp);
      A     BR;
      );
      JNB   _001;
      CALL  "HF3_W_T_B_FC54" (
           WORD1                    := #H_P_ALL_Ctrl,
           bool1                    := #H_P_ALL_Ctrl_Temp);
_001: NOP   0;
NETWORK
TITLE =
      CALL  "HF3_W_T_B_FC54" (
           WORD1                    := #IN_RD,
           bool1                    := #DI_Temp);
      NOP   0;
NETWORK
TITLE = 传递火灾报警信号
      A     DB7004.DBX 2630.0;
      =     #FireAlarm;
NETWORK
TITLE = 传递阻塞报警信号
      A     DB7004.DBX 2630.1;
      =     #BlockAlarm;
NETWORK
TITLE = 单控标志
      O     #SCtrl_Temp[0];
      O     #ALL[0];
      O     #H_P_ALL_Ctrl_Temp[3];
      S     #SFlag;
NETWORK
TITLE = 模控标志
      O     #SCtrl_Temp[1];
      O     #ALL[1];
      O     #H_P_ALL_Ctrl_Temp[4];
      O     #H_P_ALL_Ctrl_Temp[5];
      O     #FireAlarm;
      O     #BlockAlarm;
      R     #SFlag;
NETWORK
TITLE = 单/模控开
      A     #SFlag;
      A     #SCtrl_Temp[2];
      O;
      AN    #SFlag;
      A     #MCtrl[0];
      =     #Ctrl[0];
NETWORK
TITLE = 单/模控半开
      A     #SFlag;
      A     #SCtrl_Temp[3];
      O;
      AN    #SFlag;
      A     #MCtrl[1];
      =     #Ctrl[1];
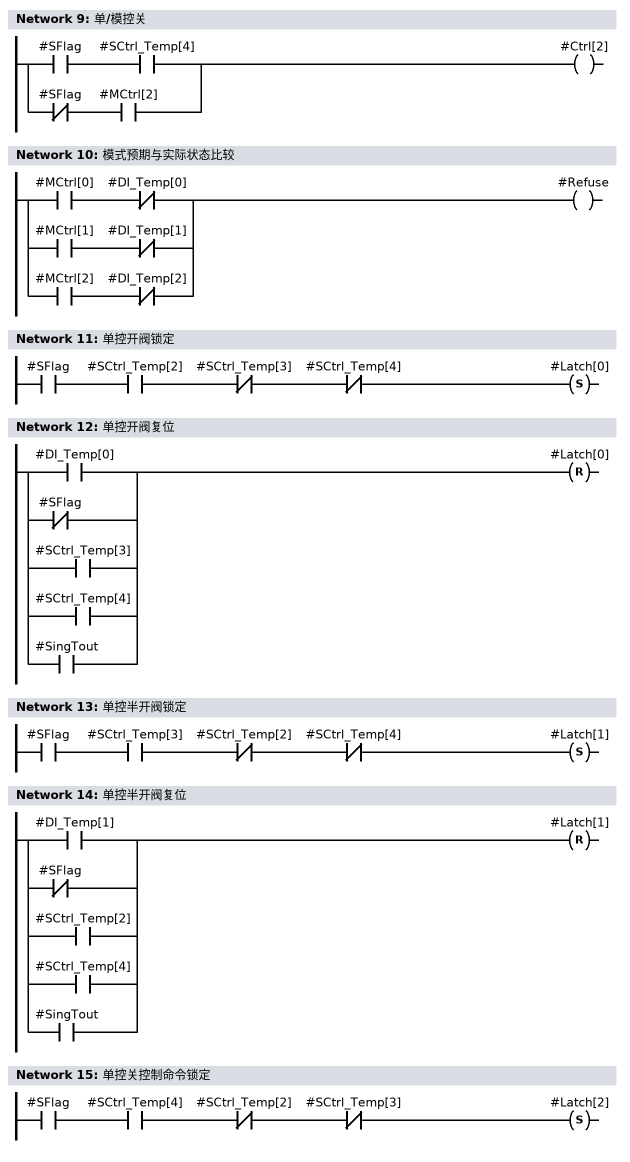
NETWORK
TITLE = 单/模控关
      A     #SFlag;
      A     #SCtrl_Temp[4];
      O;
      AN    #SFlag;
      A     #MCtrl[2];
      =     #Ctrl[2];
NETWORK
TITLE = 模式预期与实际状态比较
      A     #MCtrl[0];
      AN    #DI_Temp[0];
      O;
      A     #MCtrl[1];
      AN    #DI_Temp[1];
      O;
      A     #MCtrl[2];
      AN    #DI_Temp[2];
      =     #Refuse;
NETWORK
TITLE = 单控开阀锁定
      A     #SFlag;
      A     #SCtrl_Temp[2];
      AN    #SCtrl_Temp[3];
      AN    #SCtrl_Temp[4];
      S     #Latch[0];
NETWORK
TITLE = 单控开阀复位
      O     #DI_Temp[0];
      ON    #SFlag;
      O     #SCtrl_Temp[3];
      O     #SCtrl_Temp[4];
      O     #SingTout;
      R     #Latch[0];
NETWORK
TITLE = 单控半开阀锁定
      A     #SFlag;
      A     #SCtrl_Temp[3];
      AN    #SCtrl_Temp[2];
      AN    #SCtrl_Temp[4];
      S     #Latch[1];
NETWORK
TITLE = 单控半开阀复位
      O     #DI_Temp[1];
      ON    #SFlag;
      O     #SCtrl_Temp[2];
      O     #SCtrl_Temp[4];
      O     #SingTout;
      R     #Latch[1];
NETWORK
TITLE = 单控关控制命令锁定
      A     #SFlag;
      A     #SCtrl_Temp[4];
      AN    #SCtrl_Temp[2];
      AN    #SCtrl_Temp[3];
      S     #Latch[2];
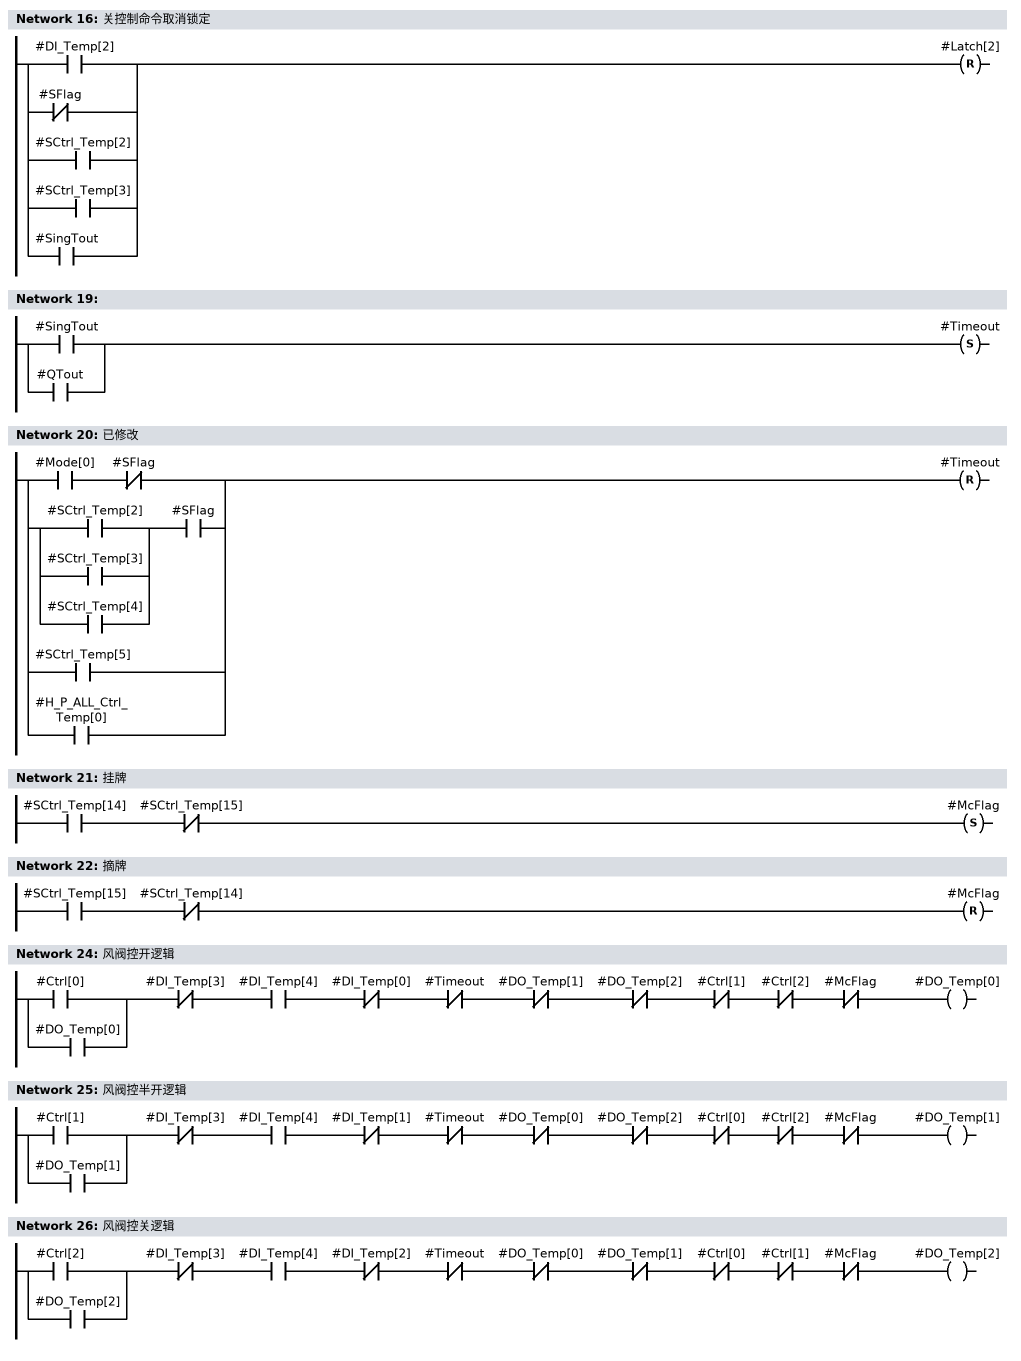
NETWORK
TITLE = 关控制命令取消锁定
      O     #DI_Temp[2];
      ON    #SFlag;
      O     #SCtrl_Temp[2];
      O     #SCtrl_Temp[3];
      O     #SingTout;
      R     #Latch[2];
NETWORK
TITLE =
      A(;
      O     #Latch[0];
      O     #Latch[1];
      O     #Latch[2];
      );
      =     L 0.0;
      BLD   103;
      BLD   16;
      =     L 7.0;
      L     DINO;
      T     LW 5;
      CDB;
      OPN   DI [LW 5];
      TAR2  LD 1;
      A     L 0.0;
      =     DIX [AR2,P#40.0];
      L     DBD [AR2,P#14.0];
      T     DID [AR2,P#42.0];
      +AR2  P#40.0;
      UC    "TON";
      LAR2  LD 1;
      A     DIX [AR2,P#46.0];
      =     DBX [AR2,P#38.4];
      CDB;
      BLD   17;
      NOP   0;
NETWORK
TITLE =
      A(;
      O     #DO_Temp[1];
      O     #DO_Temp[2];
      O     #DO_Temp[3];
      );
      =     L 0.0;
      BLD   103;
      BLD   16;
      =     L 7.0;
      L     DINO;
      T     LW 5;
      CDB;
      OPN   DI [LW 5];
      TAR2  LD 1;
      A     L 0.0;
      =     DIX [AR2,P#62.0];
      L     DBD [AR2,P#14.0];
      T     DID [AR2,P#64.0];
      +AR2  P#62.0;
      UC    "TON";
      LAR2  LD 1;
      A     DIX [AR2,P#68.0];
      =     DBX [AR2,P#38.1];
      CDB;
      BLD   17;
      NOP   0;
NETWORK
TITLE =
      O     #SingTout;
      O     #QTout;
      S     #Timeout;
NETWORK
TITLE = 已修改
      A     #Mode[0];
      AN    #SFlag;
      O;
      A(;
      O     #SCtrl_Temp[2];
      O     #SCtrl_Temp[3];
      O     #SCtrl_Temp[4];
      );
      A     #SFlag;
      O     #SCtrl_Temp[5];
      O     #H_P_ALL_Ctrl_Temp[0];
      R     #Timeout;
NETWORK
TITLE = 挂牌
      A     #SCtrl_Temp[14];
      AN    #SCtrl_Temp[15];
      S     #McFlag;
NETWORK
TITLE = 摘牌
      A     #SCtrl_Temp[15];
      AN    #SCtrl_Temp[14];
      R     #McFlag;
NETWORK
TITLE =
      A(;
      O     #DO_Temp[0];
      O     #DO_Temp[1];
      O     #DO_Temp[2];
      );
      =     L 0.0;
      BLD   103;
      BLD   16;
      =     L 7.0;
      L     DINO;
      T     LW 5;
      CDB;
      OPN   DI [LW 5];
      TAR2  LD 1;
      A     L 0.0;
      =     DIX [AR2,P#84.0];
      L     DBD [AR2,P#14.0];
      T     DID [AR2,P#86.0];
      +AR2  P#84.0;
      UC    "TON";
      LAR2  LD 1;
      A     DIX [AR2,P#90.0];
      =     DBX [AR2,P#31.2];
      CDB;
      BLD   17;
      NOP   0;
NETWORK
TITLE = 风阀控开逻辑
      A(;
      O     #Ctrl[0];
      O     #DO_Temp[0];
      );
      AN    #DI_Temp[3];
      A     #DI_Temp[4];
      AN    #DI_Temp[0];
      AN    #Timeout;
      AN    #DO_Temp[1];
      AN    #DO_Temp[2];
      AN    #Ctrl[1];
      AN    #Ctrl[2];
      AN    #McFlag;
      =     #DO_Temp[0];
NETWORK
TITLE = 风阀控半开逻辑
      A(;
      O     #Ctrl[1];
      O     #DO_Temp[1];
      );
      AN    #DI_Temp[3];
      A     #DI_Temp[4];
      AN    #DI_Temp[1];
      AN    #Timeout;
      AN    #DO_Temp[0];
      AN    #DO_Temp[2];
      AN    #Ctrl[0];
      AN    #Ctrl[2];
      AN    #McFlag;
      =     #DO_Temp[1];
NETWORK
TITLE = 风阀控关逻辑
      A(;
      O     #Ctrl[2];
      O     #DO_Temp[2];
      );
      AN    #DI_Temp[3];
      A     #DI_Temp[4];
      AN    #DI_Temp[2];
      AN    #Timeout;
      AN    #DO_Temp[0];
      AN    #DO_Temp[1];
      AN    #Ctrl[0];
      AN    #Ctrl[1];
      AN    #McFlag;
      =     #DO_Temp[2];
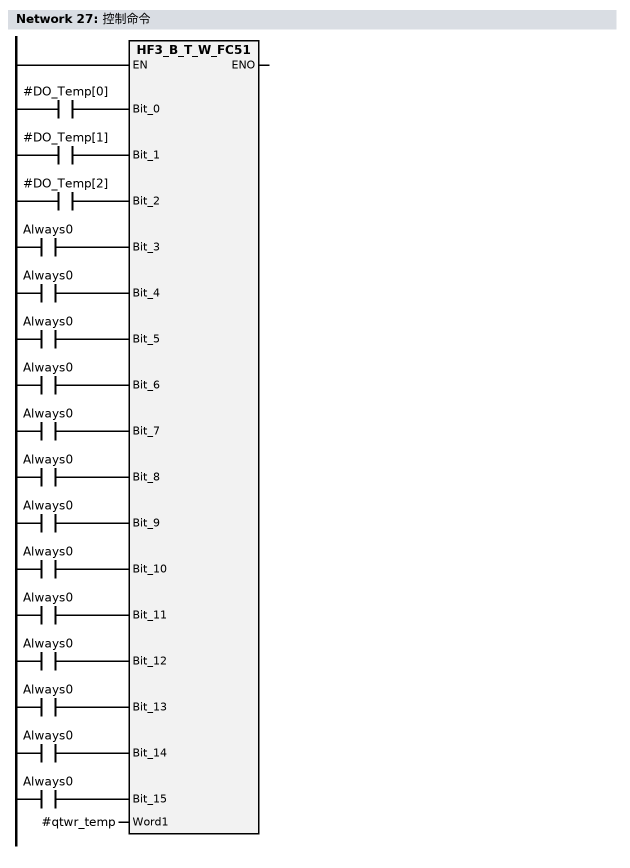
NETWORK
TITLE = 控制命令
      A     #DO_Temp[0];
      =     L 0.0;
      BLD   103;
      A     #DO_Temp[1];
      =     L 0.1;
      BLD   103;
      A     #DO_Temp[2];
      =     L 0.2;
      BLD   103;
      A     "Always0";
      =     L 0.3;
      BLD   103;
      A     "Always0";
      =     L 0.4;
      BLD   103;
      A     "Always0";
      =     L 0.5;
      BLD   103;
      A     "Always0";
      =     L 0.6;
      BLD   103;
      A     "Always0";
      =     L 0.7;
      BLD   103;
      A     "Always0";
      =     L 1.0;
      BLD   103;
      A     "Always0";
      =     L 1.1;
      BLD   103;
      A     "Always0";
      =     L 1.2;
      BLD   103;
      A     "Always0";
      =     L 1.3;
      BLD   103;
      A     "Always0";
      =     L 1.4;
      BLD   103;
      A     "Always0";
      =     L 1.5;
      BLD   103;
      A     "Always0";
      =     L 1.6;
      BLD   103;
      A     "Always0";
      =     L 1.7;
      BLD   103;
      CALL  "HF3_B_T_W_FC51" (
           Bit_0                    := L 0.0,
           Bit_1                    := L 0.1,
           Bit_2                    := L 0.2,
           Bit_3                    := L 0.3,
           Bit_4                    := L 0.4,
           Bit_5                    := L 0.5,
           Bit_6                    := L 0.6,
           Bit_7                    := L 0.7,
           Bit_8                    := L 1.0,
           Bit_9                    := L 1.1,
           Bit_10                   := L 1.2,
           Bit_11                   := L 1.3,
           Bit_12                   := L 1.4,
           Bit_13                   := L 1.5,
           Bit_14                   := L 1.6,
           Bit_15                   := L 1.7,
           Word1                    := #qtwr_temp);
      NOP   0;
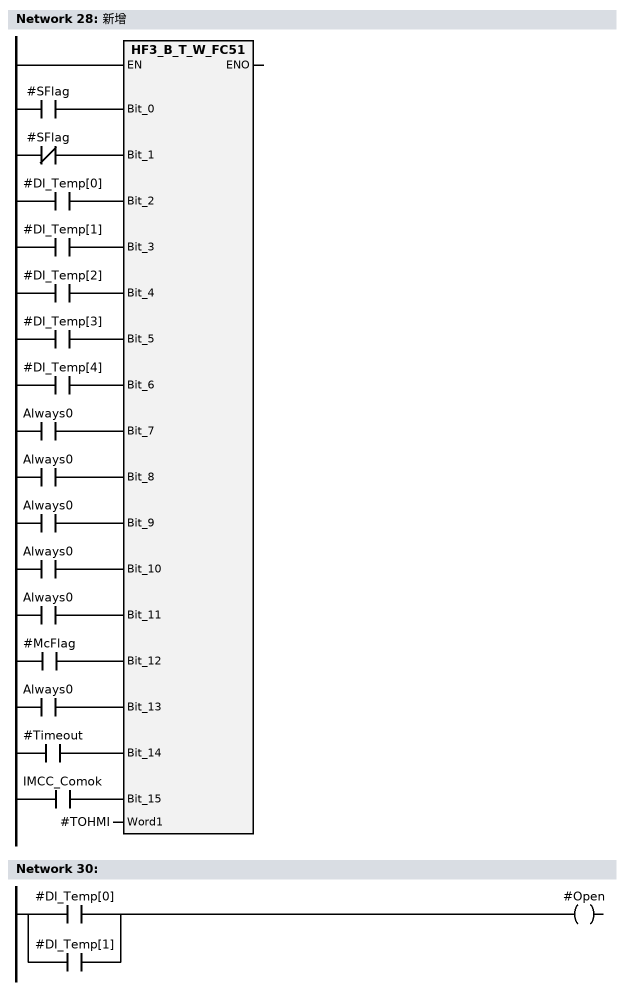
NETWORK
TITLE = 新增
      A     #SFlag;
      =     L 0.0;
      BLD   103;
      AN    #SFlag;
      =     L 0.1;
      BLD   103;
      A     #DI_Temp[0];
      =     L 0.2;
      BLD   103;
      A     #DI_Temp[1];
      =     L 0.3;
      BLD   103;
      A     #DI_Temp[2];
      =     L 0.4;
      BLD   103;
      A     #DI_Temp[3];
      =     L 0.5;
      BLD   103;
      A     #DI_Temp[4];
      =     L 0.6;
      BLD   103;
      A     "Always0";
      =     L 0.7;
      BLD   103;
      A     "Always0";
      =     L 1.0;
      BLD   103;
      A     "Always0";
      =     L 1.1;
      BLD   103;
      A     "Always0";
      =     L 1.2;
      BLD   103;
      A     "Always0";
      =     L 1.3;
      BLD   103;
      A     #McFlag;
      =     L 1.4;
      BLD   103;
      A     "Always0";
      =     L 1.5;
      BLD   103;
      A     #Timeout;
      =     L 1.6;
      BLD   103;
      A     "IMCC_Comok";
      =     L 1.7;
      BLD   103;
      CALL  "HF3_B_T_W_FC51" (
           Bit_0                    := L 0.0,
           Bit_1                    := L 0.1,
           Bit_2                    := L 0.2,
           Bit_3                    := L 0.3,
           Bit_4                    := L 0.4,
           Bit_5                    := L 0.5,
           Bit_6                    := L 0.6,
           Bit_7                    := L 0.7,
           Bit_8                    := L 1.0,
           Bit_9                    := L 1.1,
           Bit_10                   := L 1.2,
           Bit_11                   := L 1.3,
           Bit_12                   := L 1.4,
           Bit_13                   := L 1.5,
           Bit_14                   := L 1.6,
           Bit_15                   := L 1.7,
           Word1                    := #TOHMI);
      NOP   0;
NETWORK
TITLE = 参数传递
//控制命令输出
      CLR;
      L     #SCtrl;
      L     W#16#ABCD;
      <>I;
      JC    seiz;
      L     W#16#0;
      T     #qtwr_temp;
seiz: L     #qtwr_temp;
      T     #qnWR;
NETWORK
TITLE =
      O     #DI_Temp[0];
      O     #DI_Temp[1];
      =     #Open;
NETWORK
TITLE =
      SET;
      SAVE;
      CLR;
END_FUNCTION_BLOCK

FUNCTION_BLOCK "HF3_IMCC_D_FB2721"	// FB 2721
VERSION : 0.1
VAR
  PT_D : TIME  := T#45S;
  T1_D_B2 : FB 2722;
  T1_D_B5 : FB 2722;
  T2_D_B1 : FB 2722;
  T2_D_B2 : FB 2722;
  T3_D_B1 : FB 2722;
  T4_D_B1 : FB 2722;
  DM_B1 : FB 2722;
  DM_B2 : FB 2722;
  DM_B3 : FB 2722;
  DM_B4 : FB 2722;
  DM_B5 : FB 2722;
  DM_B6 : FB 2722;
  DM_B7 : FB 2722;
  DM_B8 : FB 2722;
  UOF_DT_B1 : FB 2722;
  UOF_DT_B2 : FB 2722;
  UOF_DT_B3 : FB 2722;
  UOF_DT_B4 : FB 2722;
  D_B1 : FB 2722;
  T5_D_B1 : FB 2722;
  T6_D_A1 : FB 2722;
  T6_D_A2 : FB 2722;
  T7_D_A1 : FB 2722;
  DM_A1 : FB 2722;
  DM_A2 : FB 2722;
  DM_A3 : FB 2722;
  DM_A4 : FB 2722;
  DM_A5 : FB 2722;
  DM_A6 : FB 2722;
  DM_A8 : FB 2722;
  U0F_DT_A2 : FB 2722;
  UOF_DT_A1 : FB 2722;
  UOF_DT_A3 : FB 2722;
  UOF_DT_A4 : FB 2722;
  DM_A7 : FB 2722;
END_VAR
BEGIN
NETWORK
TITLE = T6-D-A1
      A     "Always1";
      =     L 0.0;
      BLD   103;
      BLD   14;
      =     L 7.0;
      L     DINO;
      T     LW 5;
      CDB;
      OPN   DI [LW 5];
      TAR2  LD 1;
      OPN   DI 2291;
      L     DIW 610;
      OPN   DI [LW 5];
      T     DIW [AR2,P#2124.0];
      OPN   DI 6040;
      L     DIW 232;
      OPN   DI [LW 5];
      T     DIW [AR2,P#2126.0];
      OPN   DI 7005;
      L     DIW 312;
      OPN   DI [LW 5];
      T     DIW [AR2,P#2128.0];
      A     L 0.0;
      =     DIX [AR2,P#2130.0];
      BLD   11;
      L     W#16#1002;
      T     LW 10;
      L     2;
      T     LW 12;
      L     7004;
      T     LW 14;
      L     P#DBX 68.0;
      T     LD 16;
      L     W#16#1002;
      T     LW 20;
      L     2;
      T     LW 22;
      L     DINO;
      T     LW 24;
      +AR2  P#2132.0;
      TAR2;
      LAR2  LD 1;
      T     LD 26;
      UC    "BLKMOV";
      {     P#L 10.0, P#L 8.0, P#L 20.0 };
      BLD   11;
      L     W#16#1002;
      T     LW 10;
      L     2;
      T     LW 12;
      L     7005;
      T     LW 14;
      L     P#DBX 6.0;
      T     LD 16;
      L     W#16#1002;
      T     LW 20;
      L     2;
      T     LW 22;
      L     DINO;
      T     LW 24;
      +AR2  P#2134.0;
      TAR2;
      LAR2  LD 1;
      T     LD 26;
      UC    "BLKMOV";
      {     P#L 10.0, P#L 8.0, P#L 20.0 };
      BLD   11;
      L     W#16#1002;
      T     LW 10;
      L     2;
      T     LW 12;
      L     7005;
      T     LW 14;
      L     P#DBX 36.0;
      T     LD 16;
      L     W#16#1002;
      T     LW 20;
      L     2;
      T     LW 22;
      L     DINO;
      T     LW 24;
      +AR2  P#2136.0;
      TAR2;
      LAR2  LD 1;
      T     LD 26;
      UC    "BLKMOV";
      {     P#L 10.0, P#L 8.0, P#L 20.0 };
      L     DBD [AR2,P#0.0];
      T     DID [AR2,P#2138.0];
      +AR2  P#2124.0;
      UC    "HF3_IMCC_D_FB2722";
      LAR2  LD 1;
      L     DIW [AR2,P#2142.0];
      OPN   DI 2292;
      T     DIW 130;
      OPN   DI [LW 5];
      L     DIW [AR2,P#2144.0];
      OPN   DI 6004;
      T     DIW 488;
      OPN   DI [LW 5];
      A     DIX [AR2,P#2146.0];
      OPN   DI 7006;
      =     DIX 5.5;
      OPN   DI [LW 5];
      A     DIX [AR2,P#2146.1];
      OPN   DI 2555;
      =     DIX 3.6;
      OPN   DI [LW 5];
      CDB;
      BLD   15;
      NOP   0;
NETWORK
TITLE = T6-D-A2
      A     "IMCC_LOCK".T6_XPF_A1_Stop;
      =     L 0.0;
      BLD   103;
      BLD   14;
      =     L 7.0;
      L     DINO;
      T     LW 5;
      CDB;
      OPN   DI [LW 5];
      TAR2  LD 1;
      OPN   DI 2291;
      L     DIW 612;
      OPN   DI [LW 5];
      T     DIW [AR2,P#2230.0];
      OPN   DI 6040;
      L     DIW 234;
      OPN   DI [LW 5];
      T     DIW [AR2,P#2232.0];
      OPN   DI 7005;
      L     DIW 312;
      OPN   DI [LW 5];
      T     DIW [AR2,P#2234.0];
      A     L 0.0;
      =     DIX [AR2,P#2236.0];
      BLD   11;
      L     W#16#1002;
      T     LW 10;
      L     2;
      T     LW 12;
      L     7004;
      T     LW 14;
      L     P#DBX 70.0;
      T     LD 16;
      L     W#16#1002;
      T     LW 20;
      L     2;
      T     LW 22;
      L     DINO;
      T     LW 24;
      +AR2  P#2238.0;
      TAR2;
      LAR2  LD 1;
      T     LD 26;
      UC    "BLKMOV";
      {     P#L 10.0, P#L 8.0, P#L 20.0 };
      BLD   11;
      L     W#16#1002;
      T     LW 10;
      L     2;
      T     LW 12;
      L     7005;
      T     LW 14;
      L     P#DBX 6.0;
      T     LD 16;
      L     W#16#1002;
      T     LW 20;
      L     2;
      T     LW 22;
      L     DINO;
      T     LW 24;
      +AR2  P#2240.0;
      TAR2;
      LAR2  LD 1;
      T     LD 26;
      UC    "BLKMOV";
      {     P#L 10.0, P#L 8.0, P#L 20.0 };
      BLD   11;
      L     W#16#1002;
      T     LW 10;
      L     2;
      T     LW 12;
      L     7005;
      T     LW 14;
      L     P#DBX 36.0;
      T     LD 16;
      L     W#16#1002;
      T     LW 20;
      L     2;
      T     LW 22;
      L     DINO;
      T     LW 24;
      +AR2  P#2242.0;
      TAR2;
      LAR2  LD 1;
      T     LD 26;
      UC    "BLKMOV";
      {     P#L 10.0, P#L 8.0, P#L 20.0 };
      L     DBD [AR2,P#0.0];
      T     DID [AR2,P#2244.0];
      +AR2  P#2230.0;
      UC    "HF3_IMCC_D_FB2722";
      LAR2  LD 1;
      L     DIW [AR2,P#2248.0];
      OPN   DI 2292;
      T     DIW 132;
      OPN   DI [LW 5];
      L     DIW [AR2,P#2250.0];
      OPN   DI 6004;
      T     DIW 490;
      OPN   DI [LW 5];
      A     DIX [AR2,P#2252.0];
      OPN   DI 7006;
      =     DIX 5.6;
      OPN   DI [LW 5];
      A     DIX [AR2,P#2252.1];
      OPN   DI 2555;
      =     DIX 3.7;
      OPN   DI [LW 5];
      CDB;
      BLD   15;
      NOP   0;
NETWORK
TITLE = T7-D-A1
      A     "Always1";
      =     L 0.0;
      BLD   103;
      BLD   14;
      =     L 7.0;
      L     DINO;
      T     LW 5;
      CDB;
      OPN   DI [LW 5];
      TAR2  LD 1;
      OPN   DI 2291;
      L     DIW 614;
      OPN   DI [LW 5];
      T     DIW [AR2,P#2336.0];
      OPN   DI 6040;
      L     DIW 240;
      OPN   DI [LW 5];
      T     DIW [AR2,P#2338.0];
      OPN   DI 7005;
      L     DIW 312;
      OPN   DI [LW 5];
      T     DIW [AR2,P#2340.0];
      A     L 0.0;
      =     DIX [AR2,P#2342.0];
      BLD   11;
      L     W#16#1002;
      T     LW 10;
      L     2;
      T     LW 12;
      L     7004;
      T     LW 14;
      L     P#DBX 74.0;
      T     LD 16;
      L     W#16#1002;
      T     LW 20;
      L     2;
      T     LW 22;
      L     DINO;
      T     LW 24;
      +AR2  P#2344.0;
      TAR2;
      LAR2  LD 1;
      T     LD 26;
      UC    "BLKMOV";
      {     P#L 10.0, P#L 8.0, P#L 20.0 };
      BLD   11;
      L     W#16#1002;
      T     LW 10;
      L     2;
      T     LW 12;
      L     7005;
      T     LW 14;
      L     P#DBX 8.0;
      T     LD 16;
      L     W#16#1002;
      T     LW 20;
      L     2;
      T     LW 22;
      L     DINO;
      T     LW 24;
      +AR2  P#2346.0;
      TAR2;
      LAR2  LD 1;
      T     LD 26;
      UC    "BLKMOV";
      {     P#L 10.0, P#L 8.0, P#L 20.0 };
      BLD   11;
      L     W#16#1002;
      T     LW 10;
      L     2;
      T     LW 12;
      L     7005;
      T     LW 14;
      L     P#DBX 38.0;
      T     LD 16;
      L     W#16#1002;
      T     LW 20;
      L     2;
      T     LW 22;
      L     DINO;
      T     LW 24;
      +AR2  P#2348.0;
      TAR2;
      LAR2  LD 1;
      T     LD 26;
      UC    "BLKMOV";
      {     P#L 10.0, P#L 8.0, P#L 20.0 };
      L     DBD [AR2,P#0.0];
      T     DID [AR2,P#2350.0];
      +AR2  P#2336.0;
      UC    "HF3_IMCC_D_FB2722";
      LAR2  LD 1;
      L     DIW [AR2,P#2354.0];
      OPN   DI 2292;
      T     DIW 134;
      OPN   DI [LW 5];
      L     DIW [AR2,P#2356.0];
      OPN   DI 6004;
      T     DIW 492;
      OPN   DI [LW 5];
      A     DIX [AR2,P#2358.0];
      OPN   DI 7006;
      =     DIX 6.0;
      OPN   DI [LW 5];
      A     DIX [AR2,P#2358.1];
      OPN   DI 2555;
      =     DIX 4.1;
      OPN   DI [LW 5];
      CDB;
      BLD   15;
      NOP   0;
NETWORK
TITLE = DM-A1
      A     "Always1";
      =     L 0.0;
      BLD   103;
      BLD   14;
      =     L 7.0;
      L     DINO;
      T     LW 5;
      CDB;
      OPN   DI [LW 5];
      TAR2  LD 1;
      OPN   DI 2291;
      L     DIW 652;
      OPN   DI [LW 5];
      T     DIW [AR2,P#2442.0];
      OPN   DI 6040;
      L     DIW 86;
      OPN   DI [LW 5];
      T     DIW [AR2,P#2444.0];
      OPN   DI 7005;
      L     DIW 312;
      OPN   DI [LW 5];
      T     DIW [AR2,P#2446.0];
      A     L 0.0;
      =     DIX [AR2,P#2448.0];
      BLD   11;
      L     W#16#1002;
      T     LW 10;
      L     2;
      T     LW 12;
      L     7004;
      T     LW 14;
      L     P#DBX 22.0;
      T     LD 16;
      L     W#16#1002;
      T     LW 20;
      L     2;
      T     LW 22;
      L     DINO;
      T     LW 24;
      +AR2  P#2450.0;
      TAR2;
      LAR2  LD 1;
      T     LD 26;
      UC    "BLKMOV";
      {     P#L 10.0, P#L 8.0, P#L 20.0 };
      BLD   11;
      L     W#16#1002;
      T     LW 10;
      L     2;
      T     LW 12;
      L     7005;
      T     LW 14;
      L     P#DBX 2.0;
      T     LD 16;
      L     W#16#1002;
      T     LW 20;
      L     2;
      T     LW 22;
      L     DINO;
      T     LW 24;
      +AR2  P#2452.0;
      TAR2;
      LAR2  LD 1;
      T     LD 26;
      UC    "BLKMOV";
      {     P#L 10.0, P#L 8.0, P#L 20.0 };
      BLD   11;
      L     W#16#1002;
      T     LW 10;
      L     2;
      T     LW 12;
      L     7005;
      T     LW 14;
      L     P#DBX 32.0;
      T     LD 16;
      L     W#16#1002;
      T     LW 20;
      L     2;
      T     LW 22;
      L     DINO;
      T     LW 24;
      +AR2  P#2454.0;
      TAR2;
      LAR2  LD 1;
      T     LD 26;
      UC    "BLKMOV";
      {     P#L 10.0, P#L 8.0, P#L 20.0 };
      L     DBD [AR2,P#0.0];
      T     DID [AR2,P#2456.0];
      +AR2  P#2442.0;
      UC    "HF3_IMCC_D_FB2722";
      LAR2  LD 1;
      L     DIW [AR2,P#2460.0];
      OPN   DI 2292;
      T     DIW 172;
      OPN   DI [LW 5];
      L     DIW [AR2,P#2462.0];
      OPN   DI 6004;
      T     DIW 494;
      OPN   DI [LW 5];
      A     DIX [AR2,P#2464.0];
      OPN   DI 7006;
      =     DIX 3.2;
      OPN   DI [LW 5];
      CDB;
      BLD   15;
      NOP   0;
NETWORK
TITLE = DM-A2
      A     "Always1";
      =     L 0.0;
      BLD   103;
      BLD   14;
      =     L 7.0;
      L     DINO;
      T     LW 5;
      CDB;
      OPN   DI [LW 5];
      TAR2  LD 1;
      OPN   DI 2291;
      L     DIW 654;
      OPN   DI [LW 5];
      T     DIW [AR2,P#2548.0];
      OPN   DI 6040;
      L     DIW 88;
      OPN   DI [LW 5];
      T     DIW [AR2,P#2550.0];
      OPN   DI 7005;
      L     DIW 312;
      OPN   DI [LW 5];
      T     DIW [AR2,P#2552.0];
      A     L 0.0;
      =     DIX [AR2,P#2554.0];
      BLD   11;
      L     W#16#1002;
      T     LW 10;
      L     2;
      T     LW 12;
      L     7004;
      T     LW 14;
      L     P#DBX 24.0;
      T     LD 16;
      L     W#16#1002;
      T     LW 20;
      L     2;
      T     LW 22;
      L     DINO;
      T     LW 24;
      +AR2  P#2556.0;
      TAR2;
      LAR2  LD 1;
      T     LD 26;
      UC    "BLKMOV";
      {     P#L 10.0, P#L 8.0, P#L 20.0 };
      BLD   11;
      L     W#16#1002;
      T     LW 10;
      L     2;
      T     LW 12;
      L     7005;
      T     LW 14;
      L     P#DBX 2.0;
      T     LD 16;
      L     W#16#1002;
      T     LW 20;
      L     2;
      T     LW 22;
      L     DINO;
      T     LW 24;
      +AR2  P#2558.0;
      TAR2;
      LAR2  LD 1;
      T     LD 26;
      UC    "BLKMOV";
      {     P#L 10.0, P#L 8.0, P#L 20.0 };
      BLD   11;
      L     W#16#1002;
      T     LW 10;
      L     2;
      T     LW 12;
      L     7005;
      T     LW 14;
      L     P#DBX 32.0;
      T     LD 16;
      L     W#16#1002;
      T     LW 20;
      L     2;
      T     LW 22;
      L     DINO;
      T     LW 24;
      +AR2  P#2560.0;
      TAR2;
      LAR2  LD 1;
      T     LD 26;
      UC    "BLKMOV";
      {     P#L 10.0, P#L 8.0, P#L 20.0 };
      L     DBD [AR2,P#0.0];
      T     DID [AR2,P#2562.0];
      +AR2  P#2548.0;
      UC    "HF3_IMCC_D_FB2722";
      LAR2  LD 1;
      L     DIW [AR2,P#2566.0];
      OPN   DI 2292;
      T     DIW 174;
      OPN   DI [LW 5];
      L     DIW [AR2,P#2568.0];
      OPN   DI 6004;
      T     DIW 496;
      OPN   DI [LW 5];
      A     DIX [AR2,P#2570.0];
      OPN   DI 7006;
      =     DIX 3.3;
      OPN   DI [LW 5];
      CDB;
      BLD   15;
      NOP   0;
NETWORK
TITLE = DM-A3
      A     "Always1";
      =     L 0.0;
      BLD   103;
      BLD   14;
      =     L 7.0;
      L     DINO;
      T     LW 5;
      CDB;
      OPN   DI [LW 5];
      TAR2  LD 1;
      OPN   DI 2291;
      L     DIW 656;
      OPN   DI [LW 5];
      T     DIW [AR2,P#2654.0];
      OPN   DI 6040;
      L     DIW 90;
      OPN   DI [LW 5];
      T     DIW [AR2,P#2656.0];
      OPN   DI 7005;
      L     DIW 312;
      OPN   DI [LW 5];
      T     DIW [AR2,P#2658.0];
      A     L 0.0;
      =     DIX [AR2,P#2660.0];
      BLD   11;
      L     W#16#1002;
      T     LW 10;
      L     2;
      T     LW 12;
      L     7004;
      T     LW 14;
      L     P#DBX 26.0;
      T     LD 16;
      L     W#16#1002;
      T     LW 20;
      L     2;
      T     LW 22;
      L     DINO;
      T     LW 24;
      +AR2  P#2662.0;
      TAR2;
      LAR2  LD 1;
      T     LD 26;
      UC    "BLKMOV";
      {     P#L 10.0, P#L 8.0, P#L 20.0 };
      BLD   11;
      L     W#16#1002;
      T     LW 10;
      L     2;
      T     LW 12;
      L     7005;
      T     LW 14;
      L     P#DBX 2.0;
      T     LD 16;
      L     W#16#1002;
      T     LW 20;
      L     2;
      T     LW 22;
      L     DINO;
      T     LW 24;
      +AR2  P#2664.0;
      TAR2;
      LAR2  LD 1;
      T     LD 26;
      UC    "BLKMOV";
      {     P#L 10.0, P#L 8.0, P#L 20.0 };
      BLD   11;
      L     W#16#1002;
      T     LW 10;
      L     2;
      T     LW 12;
      L     7005;
      T     LW 14;
      L     P#DBX 32.0;
      T     LD 16;
      L     W#16#1002;
      T     LW 20;
      L     2;
      T     LW 22;
      L     DINO;
      T     LW 24;
      +AR2  P#2666.0;
      TAR2;
      LAR2  LD 1;
      T     LD 26;
      UC    "BLKMOV";
      {     P#L 10.0, P#L 8.0, P#L 20.0 };
      L     DBD [AR2,P#0.0];
      T     DID [AR2,P#2668.0];
      +AR2  P#2654.0;
      UC    "HF3_IMCC_D_FB2722";
      LAR2  LD 1;
      L     DIW [AR2,P#2672.0];
      OPN   DI 2292;
      T     DIW 176;
      OPN   DI [LW 5];
      L     DIW [AR2,P#2674.0];
      OPN   DI 6004;
      T     DIW 498;
      OPN   DI [LW 5];
      A     DIX [AR2,P#2676.0];
      OPN   DI 7006;
      =     DIX 3.4;
      OPN   DI [LW 5];
      CDB;
      BLD   15;
      NOP   0;
NETWORK
TITLE = DM-A4
      A     "Always1";
      =     L 0.0;
      BLD   103;
      BLD   14;
      =     L 7.0;
      L     DINO;
      T     LW 5;
      CDB;
      OPN   DI [LW 5];
      TAR2  LD 1;
      OPN   DI 2291;
      L     DIW 658;
      OPN   DI [LW 5];
      T     DIW [AR2,P#2760.0];
      OPN   DI 6040;
      L     DIW 92;
      OPN   DI [LW 5];
      T     DIW [AR2,P#2762.0];
      OPN   DI 7005;
      L     DIW 312;
      OPN   DI [LW 5];
      T     DIW [AR2,P#2764.0];
      A     L 0.0;
      =     DIX [AR2,P#2766.0];
      BLD   11;
      L     W#16#1002;
      T     LW 10;
      L     2;
      T     LW 12;
      L     7004;
      T     LW 14;
      L     P#DBX 28.0;
      T     LD 16;
      L     W#16#1002;
      T     LW 20;
      L     2;
      T     LW 22;
      L     DINO;
      T     LW 24;
      +AR2  P#2768.0;
      TAR2;
      LAR2  LD 1;
      T     LD 26;
      UC    "BLKMOV";
      {     P#L 10.0, P#L 8.0, P#L 20.0 };
      BLD   11;
      L     W#16#1002;
      T     LW 10;
      L     2;
      T     LW 12;
      L     7005;
      T     LW 14;
      L     P#DBX 2.0;
      T     LD 16;
      L     W#16#1002;
      T     LW 20;
      L     2;
      T     LW 22;
      L     DINO;
      T     LW 24;
      +AR2  P#2770.0;
      TAR2;
      LAR2  LD 1;
      T     LD 26;
      UC    "BLKMOV";
      {     P#L 10.0, P#L 8.0, P#L 20.0 };
      BLD   11;
      L     W#16#1002;
      T     LW 10;
      L     2;
      T     LW 12;
      L     7005;
      T     LW 14;
      L     P#DBX 32.0;
      T     LD 16;
      L     W#16#1002;
      T     LW 20;
      L     2;
      T     LW 22;
      L     DINO;
      T     LW 24;
      +AR2  P#2772.0;
      TAR2;
      LAR2  LD 1;
      T     LD 26;
      UC    "BLKMOV";
      {     P#L 10.0, P#L 8.0, P#L 20.0 };
      L     DBD [AR2,P#0.0];
      T     DID [AR2,P#2774.0];
      +AR2  P#2760.0;
      UC    "HF3_IMCC_D_FB2722";
      LAR2  LD 1;
      L     DIW [AR2,P#2778.0];
      OPN   DI 2292;
      T     DIW 178;
      OPN   DI [LW 5];
      L     DIW [AR2,P#2780.0];
      OPN   DI 6004;
      T     DIW 500;
      OPN   DI [LW 5];
      A     DIX [AR2,P#2782.0];
      OPN   DI 7006;
      =     DIX 3.5;
      OPN   DI [LW 5];
      CDB;
      BLD   15;
      NOP   0;
NETWORK
TITLE = DM-A5
      A     "Always1";
      =     L 0.0;
      BLD   103;
      BLD   14;
      =     L 7.0;
      L     DINO;
      T     LW 5;
      CDB;
      OPN   DI [LW 5];
      TAR2  LD 1;
      OPN   DI 2291;
      L     DIW 660;
      OPN   DI [LW 5];
      T     DIW [AR2,P#2866.0];
      OPN   DI 6040;
      L     DIW 94;
      OPN   DI [LW 5];
      T     DIW [AR2,P#2868.0];
      OPN   DI 7005;
      L     DIW 312;
      OPN   DI [LW 5];
      T     DIW [AR2,P#2870.0];
      A     L 0.0;
      =     DIX [AR2,P#2872.0];
      BLD   11;
      L     W#16#1002;
      T     LW 10;
      L     2;
      T     LW 12;
      L     7004;
      T     LW 14;
      L     P#DBX 30.0;
      T     LD 16;
      L     W#16#1002;
      T     LW 20;
      L     2;
      T     LW 22;
      L     DINO;
      T     LW 24;
      +AR2  P#2874.0;
      TAR2;
      LAR2  LD 1;
      T     LD 26;
      UC    "BLKMOV";
      {     P#L 10.0, P#L 8.0, P#L 20.0 };
      BLD   11;
      L     W#16#1002;
      T     LW 10;
      L     2;
      T     LW 12;
      L     7005;
      T     LW 14;
      L     P#DBX 2.0;
      T     LD 16;
      L     W#16#1002;
      T     LW 20;
      L     2;
      T     LW 22;
      L     DINO;
      T     LW 24;
      +AR2  P#2876.0;
      TAR2;
      LAR2  LD 1;
      T     LD 26;
      UC    "BLKMOV";
      {     P#L 10.0, P#L 8.0, P#L 20.0 };
      BLD   11;
      L     W#16#1002;
      T     LW 10;
      L     2;
      T     LW 12;
      L     7005;
      T     LW 14;
      L     P#DBX 32.0;
      T     LD 16;
      L     W#16#1002;
      T     LW 20;
      L     2;
      T     LW 22;
      L     DINO;
      T     LW 24;
      +AR2  P#2878.0;
      TAR2;
      LAR2  LD 1;
      T     LD 26;
      UC    "BLKMOV";
      {     P#L 10.0, P#L 8.0, P#L 20.0 };
      L     DBD [AR2,P#0.0];
      T     DID [AR2,P#2880.0];
      +AR2  P#2866.0;
      UC    "HF3_IMCC_D_FB2722";
      LAR2  LD 1;
      L     DIW [AR2,P#2884.0];
      OPN   DI 2292;
      T     DIW 180;
      OPN   DI [LW 5];
      L     DIW [AR2,P#2886.0];
      OPN   DI 6004;
      T     DIW 502;
      OPN   DI [LW 5];
      A     DIX [AR2,P#2888.0];
      OPN   DI 7006;
      =     DIX 3.6;
      OPN   DI [LW 5];
      CDB;
      BLD   15;
      NOP   0;
NETWORK
TITLE = DM-A6
      A     "Always1";
      =     L 0.0;
      BLD   103;
      BLD   14;
      =     L 7.0;
      L     DINO;
      T     LW 5;
      CDB;
      OPN   DI [LW 5];
      TAR2  LD 1;
      OPN   DI 2291;
      L     DIW 662;
      OPN   DI [LW 5];
      T     DIW [AR2,P#2972.0];
      OPN   DI 6040;
      L     DIW 96;
      OPN   DI [LW 5];
      T     DIW [AR2,P#2974.0];
      OPN   DI 7005;
      L     DIW 312;
      OPN   DI [LW 5];
      T     DIW [AR2,P#2976.0];
      A     L 0.0;
      =     DIX [AR2,P#2978.0];
      BLD   11;
      L     W#16#1002;
      T     LW 10;
      L     2;
      T     LW 12;
      L     7004;
      T     LW 14;
      L     P#DBX 32.0;
      T     LD 16;
      L     W#16#1002;
      T     LW 20;
      L     2;
      T     LW 22;
      L     DINO;
      T     LW 24;
      +AR2  P#2980.0;
      TAR2;
      LAR2  LD 1;
      T     LD 26;
      UC    "BLKMOV";
      {     P#L 10.0, P#L 8.0, P#L 20.0 };
      BLD   11;
      L     W#16#1002;
      T     LW 10;
      L     2;
      T     LW 12;
      L     7005;
      T     LW 14;
      L     P#DBX 2.0;
      T     LD 16;
      L     W#16#1002;
      T     LW 20;
      L     2;
      T     LW 22;
      L     DINO;
      T     LW 24;
      +AR2  P#2982.0;
      TAR2;
      LAR2  LD 1;
      T     LD 26;
      UC    "BLKMOV";
      {     P#L 10.0, P#L 8.0, P#L 20.0 };
      BLD   11;
      L     W#16#1002;
      T     LW 10;
      L     2;
      T     LW 12;
      L     7005;
      T     LW 14;
      L     P#DBX 32.0;
      T     LD 16;
      L     W#16#1002;
      T     LW 20;
      L     2;
      T     LW 22;
      L     DINO;
      T     LW 24;
      +AR2  P#2984.0;
      TAR2;
      LAR2  LD 1;
      T     LD 26;
      UC    "BLKMOV";
      {     P#L 10.0, P#L 8.0, P#L 20.0 };
      L     DBD [AR2,P#0.0];
      T     DID [AR2,P#2986.0];
      +AR2  P#2972.0;
      UC    "HF3_IMCC_D_FB2722";
      LAR2  LD 1;
      L     DIW [AR2,P#2990.0];
      OPN   DI 2292;
      T     DIW 182;
      OPN   DI [LW 5];
      L     DIW [AR2,P#2992.0];
      OPN   DI 6004;
      T     DIW 504;
      OPN   DI [LW 5];
      A     DIX [AR2,P#2994.0];
      OPN   DI 7006;
      =     DIX 3.7;
      OPN   DI [LW 5];
      CDB;
      BLD   15;
      NOP   0;
NETWORK
TITLE = DM-A7
      A     "Always1";
      =     L 0.0;
      BLD   103;
      BLD   14;
      =     L 7.0;
      L     DINO;
      T     LW 5;
      CDB;
      OPN   DI [LW 5];
      TAR2  LD 1;
      OPN   DI 2291;
      L     DIW 664;
      OPN   DI [LW 5];
      T     DIW [AR2,P#3608.0];
      OPN   DI 6040;
      L     DIW 98;
      OPN   DI [LW 5];
      T     DIW [AR2,P#3610.0];
      OPN   DI 7005;
      L     DIW 312;
      OPN   DI [LW 5];
      T     DIW [AR2,P#3612.0];
      A     L 0.0;
      =     DIX [AR2,P#3614.0];
      BLD   11;
      L     W#16#1002;
      T     LW 10;
      L     2;
      T     LW 12;
      L     7004;
      T     LW 14;
      L     P#DBX 34.0;
      T     LD 16;
      L     W#16#1002;
      T     LW 20;
      L     2;
      T     LW 22;
      L     DINO;
      T     LW 24;
      +AR2  P#3616.0;
      TAR2;
      LAR2  LD 1;
      T     LD 26;
      UC    "BLKMOV";
      {     P#L 10.0, P#L 8.0, P#L 20.0 };
      BLD   11;
      L     W#16#1002;
      T     LW 10;
      L     2;
      T     LW 12;
      L     7005;
      T     LW 14;
      L     P#DBX 2.0;
      T     LD 16;
      L     W#16#1002;
      T     LW 20;
      L     2;
      T     LW 22;
      L     DINO;
      T     LW 24;
      +AR2  P#3618.0;
      TAR2;
      LAR2  LD 1;
      T     LD 26;
      UC    "BLKMOV";
      {     P#L 10.0, P#L 8.0, P#L 20.0 };
      BLD   11;
      L     W#16#1002;
      T     LW 10;
      L     2;
      T     LW 12;
      L     7005;
      T     LW 14;
      L     P#DBX 32.0;
      T     LD 16;
      L     W#16#1002;
      T     LW 20;
      L     2;
      T     LW 22;
      L     DINO;
      T     LW 24;
      +AR2  P#3620.0;
      TAR2;
      LAR2  LD 1;
      T     LD 26;
      UC    "BLKMOV";
      {     P#L 10.0, P#L 8.0, P#L 20.0 };
      L     DBD [AR2,P#0.0];
      T     DID [AR2,P#3622.0];
      +AR2  P#3608.0;
      UC    "HF3_IMCC_D_FB2722";
      LAR2  LD 1;
      L     DIW [AR2,P#3626.0];
      OPN   DI 2292;
      T     DIW 184;
      OPN   DI [LW 5];
      L     DIW [AR2,P#3628.0];
      OPN   DI 6004;
      T     DIW 506;
      OPN   DI [LW 5];
      A     DIX [AR2,P#3630.0];
      OPN   DI 7006;
      =     DIX 4.0;
      OPN   DI [LW 5];
      CDB;
      BLD   15;
      NOP   0;
NETWORK
TITLE = DM-A8
      A     "Always1";
      =     L 0.0;
      BLD   103;
      BLD   14;
      =     L 7.0;
      L     DINO;
      T     LW 5;
      CDB;
      OPN   DI [LW 5];
      TAR2  LD 1;
      OPN   DI 2291;
      L     DIW 666;
      OPN   DI [LW 5];
      T     DIW [AR2,P#3078.0];
      OPN   DI 6040;
      L     DIW 100;
      OPN   DI [LW 5];
      T     DIW [AR2,P#3080.0];
      OPN   DI 7005;
      L     DIW 312;
      OPN   DI [LW 5];
      T     DIW [AR2,P#3082.0];
      A     L 0.0;
      =     DIX [AR2,P#3084.0];
      BLD   11;
      L     W#16#1002;
      T     LW 10;
      L     2;
      T     LW 12;
      L     7004;
      T     LW 14;
      L     P#DBX 36.0;
      T     LD 16;
      L     W#16#1002;
      T     LW 20;
      L     2;
      T     LW 22;
      L     DINO;
      T     LW 24;
      +AR2  P#3086.0;
      TAR2;
      LAR2  LD 1;
      T     LD 26;
      UC    "BLKMOV";
      {     P#L 10.0, P#L 8.0, P#L 20.0 };
      BLD   11;
      L     W#16#1002;
      T     LW 10;
      L     2;
      T     LW 12;
      L     7005;
      T     LW 14;
      L     P#DBX 2.0;
      T     LD 16;
      L     W#16#1002;
      T     LW 20;
      L     2;
      T     LW 22;
      L     DINO;
      T     LW 24;
      +AR2  P#3088.0;
      TAR2;
      LAR2  LD 1;
      T     LD 26;
      UC    "BLKMOV";
      {     P#L 10.0, P#L 8.0, P#L 20.0 };
      BLD   11;
      L     W#16#1002;
      T     LW 10;
      L     2;
      T     LW 12;
      L     7005;
      T     LW 14;
      L     P#DBX 32.0;
      T     LD 16;
      L     W#16#1002;
      T     LW 20;
      L     2;
      T     LW 22;
      L     DINO;
      T     LW 24;
      +AR2  P#3090.0;
      TAR2;
      LAR2  LD 1;
      T     LD 26;
      UC    "BLKMOV";
      {     P#L 10.0, P#L 8.0, P#L 20.0 };
      L     DBD [AR2,P#0.0];
      T     DID [AR2,P#3092.0];
      +AR2  P#3078.0;
      UC    "HF3_IMCC_D_FB2722";
      LAR2  LD 1;
      L     DIW [AR2,P#3096.0];
      OPN   DI 2292;
      T     DIW 186;
      OPN   DI [LW 5];
      L     DIW [AR2,P#3098.0];
      OPN   DI 6004;
      T     DIW 508;
      OPN   DI [LW 5];
      A     DIX [AR2,P#3100.0];
      OPN   DI 7006;
      =     DIX 4.1;
      OPN   DI [LW 5];
      A     DIX [AR2,P#3100.1];
      OPN   DI 2555;
      =     DIX 2.2;
      OPN   DI [LW 5];
      CDB;
      BLD   15;
      NOP   0;
END_FUNCTION_BLOCK

FUNCTION_BLOCK "HF3_IMCC_D_FB2722"	// FB 2722
VERSION : 0.1
VAR_INPUT
  IN_RD : WORD ;
  SCtrl : WORD ;	//控制命令
  H_P_ALL_Ctrl : WORD ;	//全局命令
  Stop : BOOL ;	//连锁信号
  MCtrl : ARRAY  [0 .. 3 ] OF //0-开阀1-关阀
  BOOL ;
  Mode : ARRAY  [0 .. 15 ] OF //0-开始1-结束2-执行中
  BOOL ;
  ALL : ARRAY  [0 .. 15 ] OF //单系统命令
  BOOL ;
  PT : TIME ;	//设备动作超时
END_VAR
VAR_OUTPUT
  qnWR : WORD ;	//阀控制信息
  ToHMI : WORD ;	//给上位信号
  Refuse : BOOL ;	//模式不符
  Open : BOOL ;	//阀控制信息
END_VAR
VAR
  qtwr_temp : WORD ;
  SCtrl_Temp : ARRAY  [0 .. 15 ] OF //01-单模23-开关
  BOOL ;
  DI_Temp : ARRAY  [0 .. 15 ] OF //23-开关
  BOOL ;
  DO_Temp : ARRAY  [0 .. 15 ] OF //1-开2-关输出
  BOOL ;
  H_P_ALL_Ctrl_Temp : ARRAY  [0 .. 15 ] OF BOOL ;
  Ctrl : ARRAY  [0 .. 15 ] OF //01-开关
  BOOL ;
  Latch : ARRAY  [0 .. 15 ] OF //控制锁定
  BOOL ;
  SFlag : BOOL ;	//单控标志
  QTout : BOOL ;
  Timeout : BOOL ;	//设备动作超时
  McFlag : BOOL ;	//检修牌
  SIngTout : BOOL ;
  FireAlarm : BOOL ;	//火灾信号
  BlockAlarm : BOOL ;	//阻塞信号
  Ton1 : SFB 4;
  Ton2 : SFB 4;
  Ton3 : SFB 4;
END_VAR
BEGIN
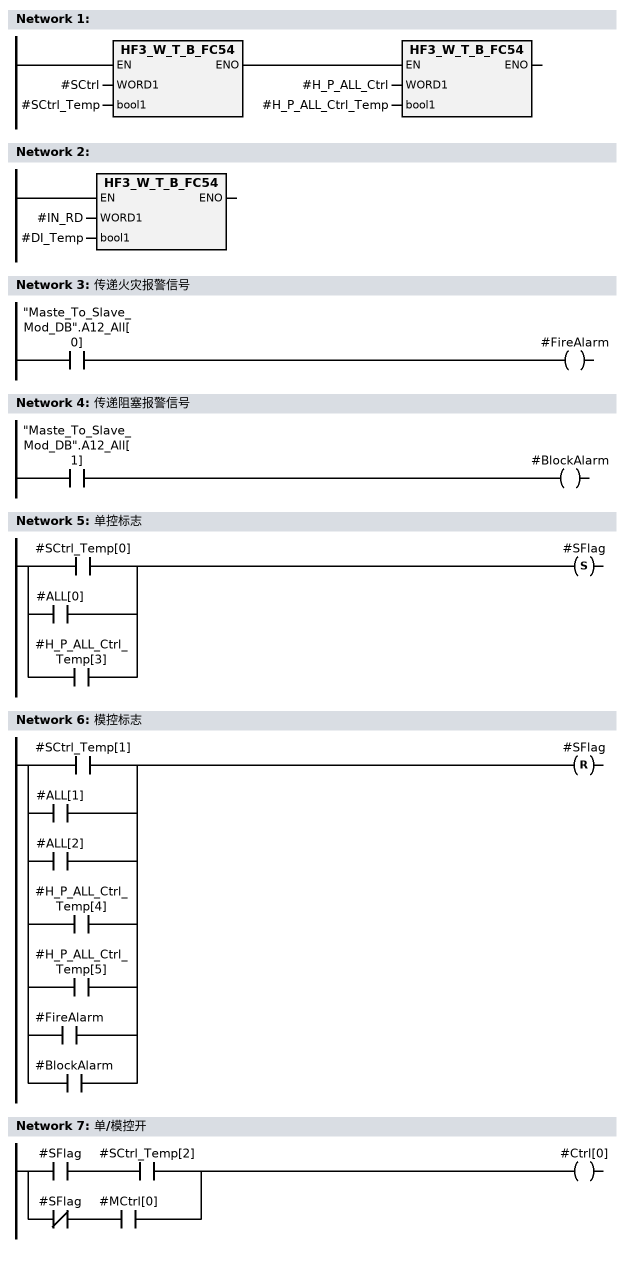
NETWORK
TITLE =
      A(;
      CALL  "HF3_W_T_B_FC54" (
           WORD1                    := #SCtrl,
           bool1                    := #SCtrl_Temp);
      A     BR;
      );
      JNB   _001;
      CALL  "HF3_W_T_B_FC54" (
           WORD1                    := #H_P_ALL_Ctrl,
           bool1                    := #H_P_ALL_Ctrl_Temp);
_001: NOP   0;
NETWORK
TITLE =
      CALL  "HF3_W_T_B_FC54" (
           WORD1                    := #IN_RD,
           bool1                    := #DI_Temp);
      NOP   0;
NETWORK
TITLE = 传递火灾报警信号
      A     "Maste_To_Slave_Mod_DB".A12_All[0];
      =     #FireAlarm;
NETWORK
TITLE = 传递阻塞报警信号
      A     "Maste_To_Slave_Mod_DB".A12_All[1];
      =     #BlockAlarm;
NETWORK
TITLE = 单控标志
      O     #SCtrl_Temp[0];
      O     #ALL[0];
      O     #H_P_ALL_Ctrl_Temp[3];
      S     #SFlag;
NETWORK
TITLE = 模控标志
      O     #SCtrl_Temp[1];
      O     #ALL[1];
      O     #ALL[2];
      O     #H_P_ALL_Ctrl_Temp[4];
      O     #H_P_ALL_Ctrl_Temp[5];
      O     #FireAlarm;
      O     #BlockAlarm;
      R     #SFlag;
NETWORK
TITLE = 单/模控开
      A     #SFlag;
      A     #SCtrl_Temp[2];
      O;
      AN    #SFlag;
      A     #MCtrl[0];
      =     #Ctrl[0];
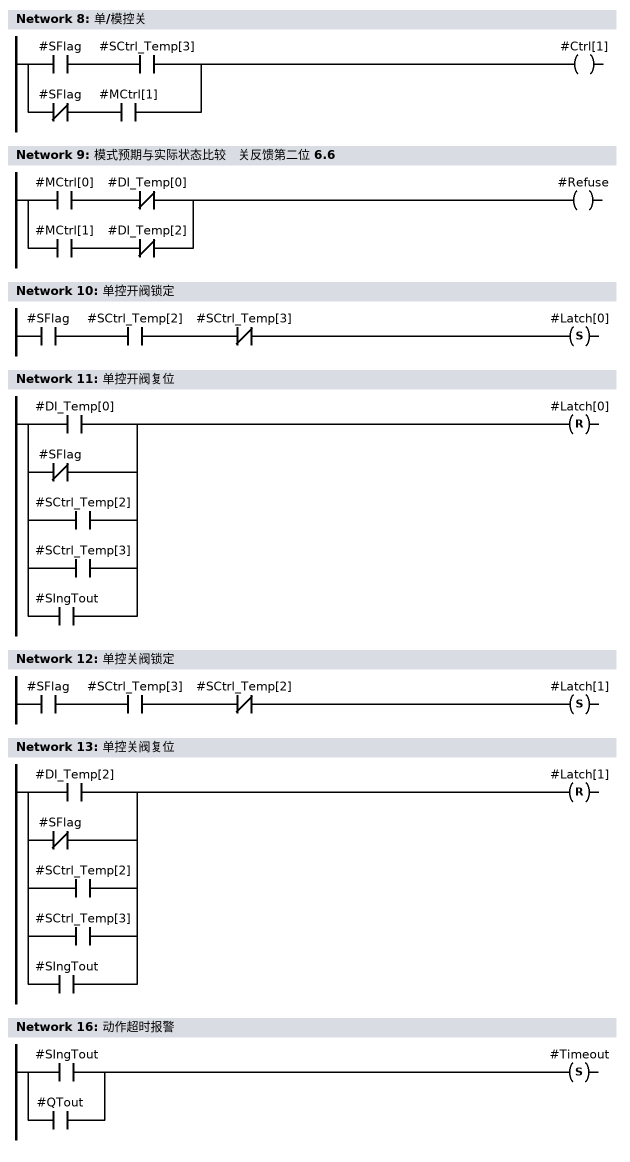
NETWORK
TITLE = 单/模控关
      A     #SFlag;
      A     #SCtrl_Temp[3];
      O;
      AN    #SFlag;
      A     #MCtrl[1];
      =     #Ctrl[1];
NETWORK
TITLE = 模式预期与实际状态比较   关反馈第二位 6.6
      A     #MCtrl[0];
      AN    #DI_Temp[0];
      O;
      A     #MCtrl[1];
      AN    #DI_Temp[2];
      =     #Refuse;
NETWORK
TITLE = 单控开阀锁定
      A     #SFlag;
      A     #SCtrl_Temp[2];
      AN    #SCtrl_Temp[3];
      S     #Latch[0];
NETWORK
TITLE = 单控开阀复位
      O     #DI_Temp[0];
      ON    #SFlag;
      O     #SCtrl_Temp[2];
      O     #SCtrl_Temp[3];
      O     #SIngTout;
      R     #Latch[0];
NETWORK
TITLE = 单控关阀锁定
      A     #SFlag;
      A     #SCtrl_Temp[3];
      AN    #SCtrl_Temp[2];
      S     #Latch[1];
NETWORK
TITLE = 单控关阀复位
      O     #DI_Temp[2];
      ON    #SFlag;
      O     #SCtrl_Temp[2];
      O     #SCtrl_Temp[3];
      O     #SIngTout;
      R     #Latch[1];
NETWORK
TITLE = 控开超时
      A(;
      O     #Latch[0];
      O     #Latch[1];
      );
      =     L 0.0;
      BLD   103;
      BLD   16;
      =     L 7.0;
      L     DINO;
      T     LW 5;
      CDB;
      OPN   DI [LW 5];
      TAR2  LD 1;
      A     L 0.0;
      =     DIX [AR2,P#40.0];
      L     DBD [AR2,P#14.0];
      T     DID [AR2,P#42.0];
      +AR2  P#40.0;
      UC    "TON";
      LAR2  LD 1;
      A     DIX [AR2,P#46.0];
      =     DBX [AR2,P#38.4];
      CDB;
      BLD   17;
      NOP   0;
NETWORK
TITLE = 控关超时
      A(;
      O     #DO_Temp[1];
      O     #DO_Temp[2];
      );
      =     L 0.0;
      BLD   103;
      BLD   16;
      =     L 7.0;
      L     DINO;
      T     LW 5;
      CDB;
      OPN   DI [LW 5];
      TAR2  LD 1;
      A     L 0.0;
      =     DIX [AR2,P#62.0];
      L     DBD [AR2,P#14.0];
      T     DID [AR2,P#64.0];
      +AR2  P#62.0;
      UC    "TON";
      LAR2  LD 1;
      A     DIX [AR2,P#68.0];
      =     DBX [AR2,P#38.1];
      CDB;
      BLD   17;
      NOP   0;
NETWORK
TITLE = 动作超时报警
      O     #SIngTout;
      O     #QTout;
      S     #Timeout;
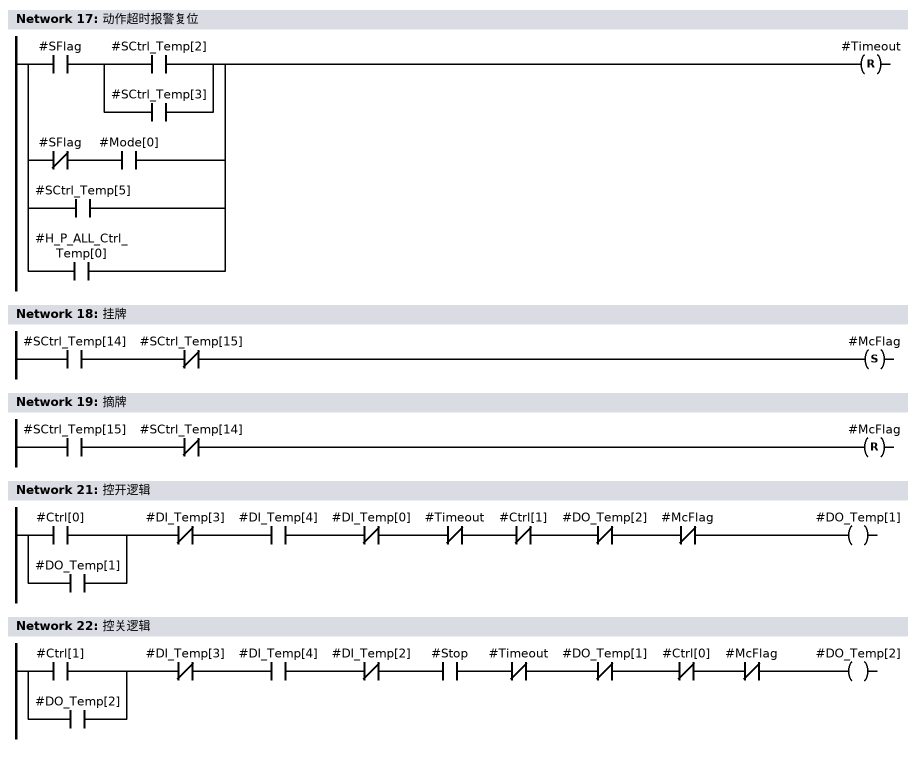
NETWORK
TITLE = 动作超时报警复位
      A     #SFlag;
      A(;
      O     #SCtrl_Temp[2];
      O     #SCtrl_Temp[3];
      );
      O;
      AN    #SFlag;
      A     #Mode[0];
      O     #SCtrl_Temp[5];
      O     #H_P_ALL_Ctrl_Temp[0];
      R     #Timeout;
NETWORK
TITLE = 挂牌
      A     #SCtrl_Temp[14];
      AN    #SCtrl_Temp[15];
      S     #McFlag;
NETWORK
TITLE = 摘牌
      A     #SCtrl_Temp[15];
      AN    #SCtrl_Temp[14];
      R     #McFlag;
NETWORK
TITLE =
      A(;
      O     #DO_Temp[1];
      O     #DO_Temp[2];
      );
      =     L 0.0;
      BLD   103;
      BLD   16;
      =     L 7.0;
      L     DINO;
      T     LW 5;
      CDB;
      OPN   DI [LW 5];
      TAR2  LD 1;
      A     L 0.0;
      =     DIX [AR2,P#84.0];
      L     L#20000;
      T     DID [AR2,P#86.0];
      +AR2  P#84.0;
      UC    "TON";
      LAR2  LD 1;
      A     DIX [AR2,P#90.0];
      =     DBX [AR2,P#31.2];
      CDB;
      BLD   17;
      NOP   0;
NETWORK
TITLE = 控开逻辑
      A(;
      O     #Ctrl[0];
      O     #DO_Temp[1];
      );
      AN    #DI_Temp[3];
      A     #DI_Temp[4];
      AN    #DI_Temp[0];
      AN    #Timeout;
      AN    #Ctrl[1];
      AN    #DO_Temp[2];
      AN    #McFlag;
      =     #DO_Temp[1];
NETWORK
TITLE = 控关逻辑
      A(;
      O     #Ctrl[1];
      O     #DO_Temp[2];
      );
      AN    #DI_Temp[3];
      A     #DI_Temp[4];
      AN    #DI_Temp[2];
      A     #Stop;
      AN    #Timeout;
      AN    #DO_Temp[1];
      AN    #Ctrl[0];
      AN    #McFlag;
      =     #DO_Temp[2];
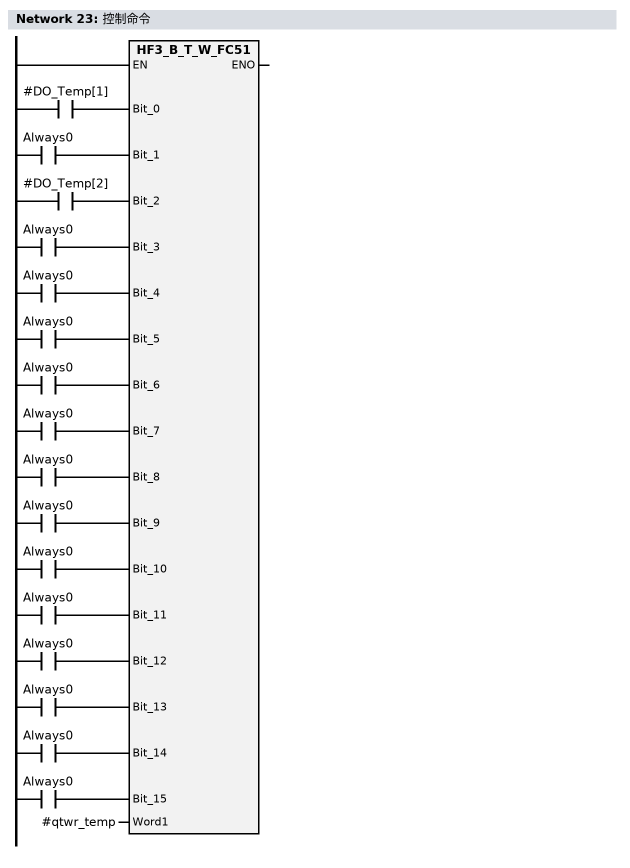
NETWORK
TITLE = 控制命令
      A     #DO_Temp[1];
      =     L 0.0;
      BLD   103;
      A     "Always0";
      =     L 0.1;
      BLD   103;
      A     #DO_Temp[2];
      =     L 0.2;
      BLD   103;
      A     "Always0";
      =     L 0.3;
      BLD   103;
      A     "Always0";
      =     L 0.4;
      BLD   103;
      A     "Always0";
      =     L 0.5;
      BLD   103;
      A     "Always0";
      =     L 0.6;
      BLD   103;
      A     "Always0";
      =     L 0.7;
      BLD   103;
      A     "Always0";
      =     L 1.0;
      BLD   103;
      A     "Always0";
      =     L 1.1;
      BLD   103;
      A     "Always0";
      =     L 1.2;
      BLD   103;
      A     "Always0";
      =     L 1.3;
      BLD   103;
      A     "Always0";
      =     L 1.4;
      BLD   103;
      A     "Always0";
      =     L 1.5;
      BLD   103;
      A     "Always0";
      =     L 1.6;
      BLD   103;
      A     "Always0";
      =     L 1.7;
      BLD   103;
      CALL  "HF3_B_T_W_FC51" (
           Bit_0                    := L 0.0,
           Bit_1                    := L 0.1,
           Bit_2                    := L 0.2,
           Bit_3                    := L 0.3,
           Bit_4                    := L 0.4,
           Bit_5                    := L 0.5,
           Bit_6                    := L 0.6,
           Bit_7                    := L 0.7,
           Bit_8                    := L 1.0,
           Bit_9                    := L 1.1,
           Bit_10                   := L 1.2,
           Bit_11                   := L 1.3,
           Bit_12                   := L 1.4,
           Bit_13                   := L 1.5,
           Bit_14                   := L 1.6,
           Bit_15                   := L 1.7,
           Word1                    := #qtwr_temp);
      NOP   0;
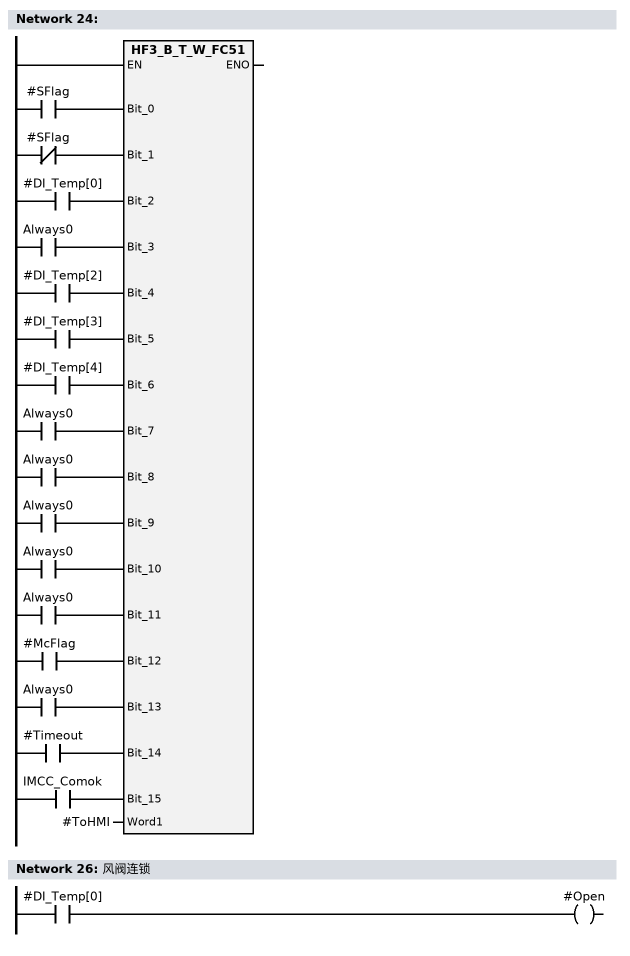
NETWORK
TITLE =
      A     #SFlag;
      =     L 0.0;
      BLD   103;
      AN    #SFlag;
      =     L 0.1;
      BLD   103;
      A     #DI_Temp[0];
      =     L 0.2;
      BLD   103;
      A     "Always0";
      =     L 0.3;
      BLD   103;
      A     #DI_Temp[2];
      =     L 0.4;
      BLD   103;
      A     #DI_Temp[3];
      =     L 0.5;
      BLD   103;
      A     #DI_Temp[4];
      =     L 0.6;
      BLD   103;
      A     "Always0";
      =     L 0.7;
      BLD   103;
      A     "Always0";
      =     L 1.0;
      BLD   103;
      A     "Always0";
      =     L 1.1;
      BLD   103;
      A     "Always0";
      =     L 1.2;
      BLD   103;
      A     "Always0";
      =     L 1.3;
      BLD   103;
      A     #McFlag;
      =     L 1.4;
      BLD   103;
      A     "Always0";
      =     L 1.5;
      BLD   103;
      A     #Timeout;
      =     L 1.6;
      BLD   103;
      A     "IMCC_Comok";
      =     L 1.7;
      BLD   103;
      CALL  "HF3_B_T_W_FC51" (
           Bit_0                    := L 0.0,
           Bit_1                    := L 0.1,
           Bit_2                    := L 0.2,
           Bit_3                    := L 0.3,
           Bit_4                    := L 0.4,
           Bit_5                    := L 0.5,
           Bit_6                    := L 0.6,
           Bit_7                    := L 0.7,
           Bit_8                    := L 1.0,
           Bit_9                    := L 1.1,
           Bit_10                   := L 1.2,
           Bit_11                   := L 1.3,
           Bit_12                   := L 1.4,
           Bit_13                   := L 1.5,
           Bit_14                   := L 1.6,
           Bit_15                   := L 1.7,
           Word1                    := #ToHMI);
      NOP   0;
NETWORK
TITLE = 控制命令传递
//控制命令输出
      CLR;
      L     #SCtrl;
      L     W#16#ABCD;
      <>I;
      JC    seiz;
      L     W#16#0;
      T     #qtwr_temp;
seiz: L     #qtwr_temp;
      T     #qnWR;
NETWORK
TITLE = 风阀连锁
      A     #DI_Temp[0];
      =     #Open;
NETWORK
TITLE =
      SET;
      SAVE;
      CLR;
END_FUNCTION_BLOCK

FUNCTION_BLOCK "HF3_JH_YC_FB2731"	// FB 2731
TITLE = 电子净化装置-压差报警打包上传综合监控
VERSION : 0.1
BEGIN
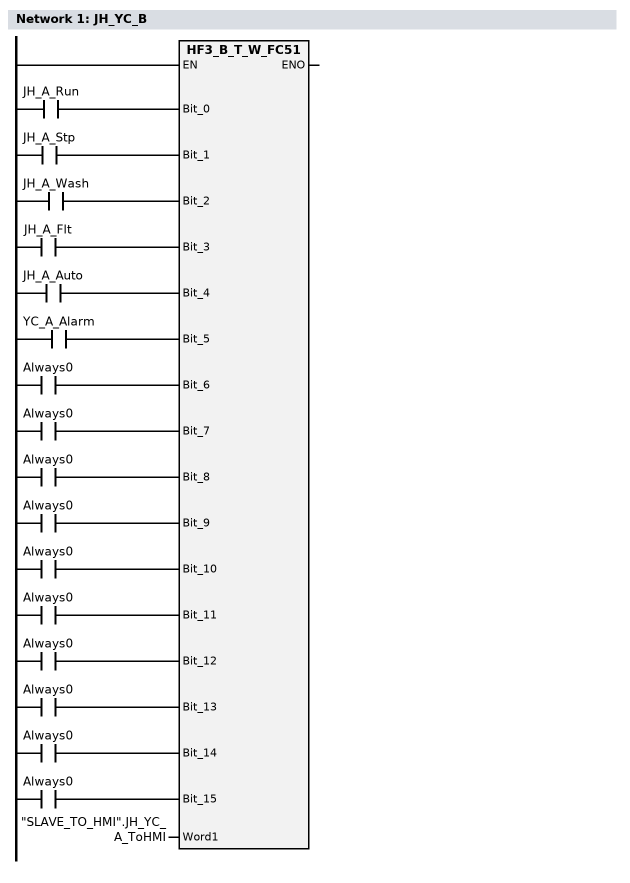
NETWORK
TITLE = JH_YC_B
      A     "JH_A_Run";
      =     L 0.0;
      BLD   103;
      A     "JH_A_Stp";
      =     L 0.1;
      BLD   103;
      A     "JH_A_Wash";
      =     L 0.2;
      BLD   103;
      A     "JH_A_Flt";
      =     L 0.3;
      BLD   103;
      A     "JH_A_Auto";
      =     L 0.4;
      BLD   103;
      A     "YC_A_Alarm";
      =     L 0.5;
      BLD   103;
      A     "Always0";
      =     L 0.6;
      BLD   103;
      A     "Always0";
      =     L 0.7;
      BLD   103;
      A     "Always0";
      =     L 1.0;
      BLD   103;
      A     "Always0";
      =     L 1.1;
      BLD   103;
      A     "Always0";
      =     L 1.2;
      BLD   103;
      A     "Always0";
      =     L 1.3;
      BLD   103;
      A     "Always0";
      =     L 1.4;
      BLD   103;
      A     "Always0";
      =     L 1.5;
      BLD   103;
      A     "Always0";
      =     L 1.6;
      BLD   103;
      A     "Always0";
      =     L 1.7;
      BLD   103;
      CALL  "HF3_B_T_W_FC51" (
           Bit_0                    := L 0.0,
           Bit_1                    := L 0.1,
           Bit_2                    := L 0.2,
           Bit_3                    := L 0.3,
           Bit_4                    := L 0.4,
           Bit_5                    := L 0.5,
           Bit_6                    := L 0.6,
           Bit_7                    := L 0.7,
           Bit_8                    := L 1.0,
           Bit_9                    := L 1.1,
           Bit_10                   := L 1.2,
           Bit_11                   := L 1.3,
           Bit_12                   := L 1.4,
           Bit_13                   := L 1.5,
           Bit_14                   := L 1.6,
           Bit_15                   := L 1.7,
           Word1                    := "SLAVE_TO_HMI".JH_YC_A_ToHMI);
      NOP   0;
END_FUNCTION_BLOCK

FUNCTION_BLOCK "HF3_DPH_FB2751"	// FB 2751
//AN_K1_DPF_A1_SCtrl:WORD := 16#00;
//AN_DPF_A1_SCtrl:WORD := 16#00;
//AN_K3_DPF_A1_SCtrl:WORD := 16#00;
//AN_K2_DPF_A1_SCtrl:WORD := 16#00;
//
VERSION : 0.1
VAR
  PT_DPH : TIME  := T#45S;
  SDPH_B2 : FB 2752;
  SDPH_K1_B1 : FB 2752;
  SDPH_K2_B1 : FB 2752;
  SDPH_K3_B1 : FB 2752;
  SDPF_K2_B1 : FB 2752;
  DPH_A1 : FB 2752;
  DPH_K4_A1 : FB 2752;
END_VAR
BEGIN
NETWORK
TITLE = SDPH_B1
      A     "SDPH_K4_A1_LR";
      =     L 0.0;
      BLD   103;
      A     "Maste_To_Slave_Mod_DB".FireAlarm;
      =     L 0.1;
      BLD   103;
      BLD   14;
      =     L 7.0;
      L     DINO;
      T     LW 5;
      CDB;
      OPN   DI [LW 5];
      TAR2  LD 1;
      OPN   DI 6003;
      L     DIW 2;
      OPN   DI [LW 5];
      T     DIW [AR2,P#1164.0];
      A     L 0.0;
      =     DIX [AR2,P#1166.0];
      L     "SDPH_A_aiPFB";
      T     DIW [AR2,P#1168.0];
      OPN   DI 6003;
      L     DIW 446;
      OPN   DI [LW 5];
      T     DIW [AR2,P#1170.0];
      OPN   DI 6003;
      L     DIW 448;
      OPN   DI [LW 5];
      T     DIW [AR2,P#1172.0];
      OPN   DI 6003;
      L     DIW 450;
      OPN   DI [LW 5];
      T     DIW [AR2,P#1174.0];
      L     DBD [AR2,P#0.0];
      T     DID [AR2,P#1182.0];
      OPN   DI 7005;
      L     DIW 312;
      OPN   DI [LW 5];
      T     DIW [AR2,P#1188.0];
      A     L 0.1;
      =     DIX [AR2,P#1190.0];
      OPN   DI 6003;
      L     DIW 452;
      OPN   DI [LW 5];
      T     DIW [AR2,P#1192.0];
      +AR2  P#1164.0;
      UC    "HF3_DPH_FB2752";
      LAR2  LD 1;
      L     DIW [AR2,P#1196.0];
      OPN   DI 6004;
      T     DIW 0;
      OPN   DI [LW 5];
      L     DIW [AR2,P#1198.0];
      T     "SDPH_K4_A1_aqPset";
      L     DID [AR2,P#1200.0];
      OPN   DI 6004;
      T     DID 2;
      OPN   DI [LW 5];
      CDB;
      BLD   15;
      NOP   0;
NETWORK
TITLE = SDPH-K4-A1
      A     "SDPH_A1_LR";
      =     L 0.0;
      BLD   103;
      A     "Maste_To_Slave_Mod_DB".FireAlarm;
      =     L 0.1;
      BLD   103;
      BLD   14;
      =     L 7.0;
      L     DINO;
      T     LW 5;
      CDB;
      OPN   DI [LW 5];
      TAR2  LD 1;
      OPN   DI 6003;
      L     DIW 0;
      OPN   DI [LW 5];
      T     DIW [AR2,P#1396.0];
      A     L 0.0;
      =     DIX [AR2,P#1398.0];
      L     "SDPH_K4_A1_aiPFB";
      T     DIW [AR2,P#1400.0];
      OPN   DI 6003;
      L     DIW 438;
      OPN   DI [LW 5];
      T     DIW [AR2,P#1402.0];
      OPN   DI 6003;
      L     DIW 440;
      OPN   DI [LW 5];
      T     DIW [AR2,P#1404.0];
      OPN   DI 6003;
      L     DIW 442;
      OPN   DI [LW 5];
      T     DIW [AR2,P#1406.0];
      L     DBD [AR2,P#0.0];
      T     DID [AR2,P#1414.0];
      OPN   DI 7005;
      L     DIW 312;
      OPN   DI [LW 5];
      T     DIW [AR2,P#1420.0];
      A     L 0.1;
      =     DIX [AR2,P#1422.0];
      OPN   DI 6003;
      L     DIW 444;
      OPN   DI [LW 5];
      T     DIW [AR2,P#1424.0];
      +AR2  P#1396.0;
      UC    "HF3_DPH_FB2752";
      LAR2  LD 1;
      L     DIW [AR2,P#1428.0];
      OPN   DI 6004;
      T     DIW 6;
      OPN   DI [LW 5];
      L     DIW [AR2,P#1430.0];
      T     "SDPH_A1_aqPset";
      L     DID [AR2,P#1432.0];
      OPN   DI 6004;
      T     DID 8;
      OPN   DI [LW 5];
      CDB;
      BLD   15;
      NOP   0;
END_FUNCTION_BLOCK

FUNCTION_BLOCK "HF3_DPH_FB2752"	// FB 2752
//pid
//
VERSION : 0.1
VAR_INPUT
  SCtrl : WORD ;	//[0]单控[1]模控[2]PID使能[3]PID非使能[14]挂检修牌[15]摘检修牌
  SDF_DI_LR : BOOL ;	//远程/就地
  aiValFB : INT ;	//开度反馈
  Kp : INT ;	//Kp值设定
  Ki : INT ;	//Ki值设定
  SP : INT ;	//目标设定值(SP)设定
  PV : INT ;	//反馈温度
  MCtrl : ARRAY  [0 .. 3 ] OF BOOL ;
  Mode : ARRAY  [0 .. 15 ] OF BOOL ;
  PT : TIME ;
  ALL : ARRAY  [0 .. 15 ] OF //单系统控制
  BOOL ;
  H_P_All_Ctrl : WORD ;	//全局命令
  FireAlarm : BOOL ;	//火灾信号
  ManuSet : INT ;	//手动开度设定
  Fit : BOOL ;
END_VAR
VAR_OUTPUT
  ToHMI : WORD ;	//[0]单控标志，[1]模控标志，[2]模式开阀，[3]模式开阀，[4]PID使能，[12]挂牌，[14]
  aqValSet : INT ;	//开度控制
  ValveFB : REAL ;	//阀门开度反馈
  ActSet : INT ;	//实际阀位设定
END_VAR
VAR
  SFlag : BOOL ;	//单控标志
  lr : BOOL ;	//远程/就地
  realAQ : REAL ;	//AQ的浮点输出
  Timeout : BOOL ;
  MAN_AUTO : BOOL ;	//手自动
  McFlag : BOOL ;	//检修牌
  SCtrl_Temp : ARRAY  [0 .. 15 ] OF //HMI控制
  BOOL ;
  PID_EN : BOOL ;	//pid使能
  ManuSet1 : INT ;
  h_p_all_temp : ARRAY  [0 .. 15 ] OF BOOL ;
  ton1 : SFB 4;
  singout : BOOL ;	//单控超时
  tr_s : BOOL ;
  tr_i : REAL ;
  manuset1_temp : DINT ;
  real_temp : REAL ;
  div_out : REAL ;
  pi : FB 41;
  DINT_TEMP_1 : DINT ;
  OMS_REAL : REAL ;
END_VAR
VAR_TEMP
  sub_temp : INT ;
  ABS_TEMP : INT ;
  end : BOOL ;
  WORD_TEMP1 : WORD ;
END_VAR
BEGIN
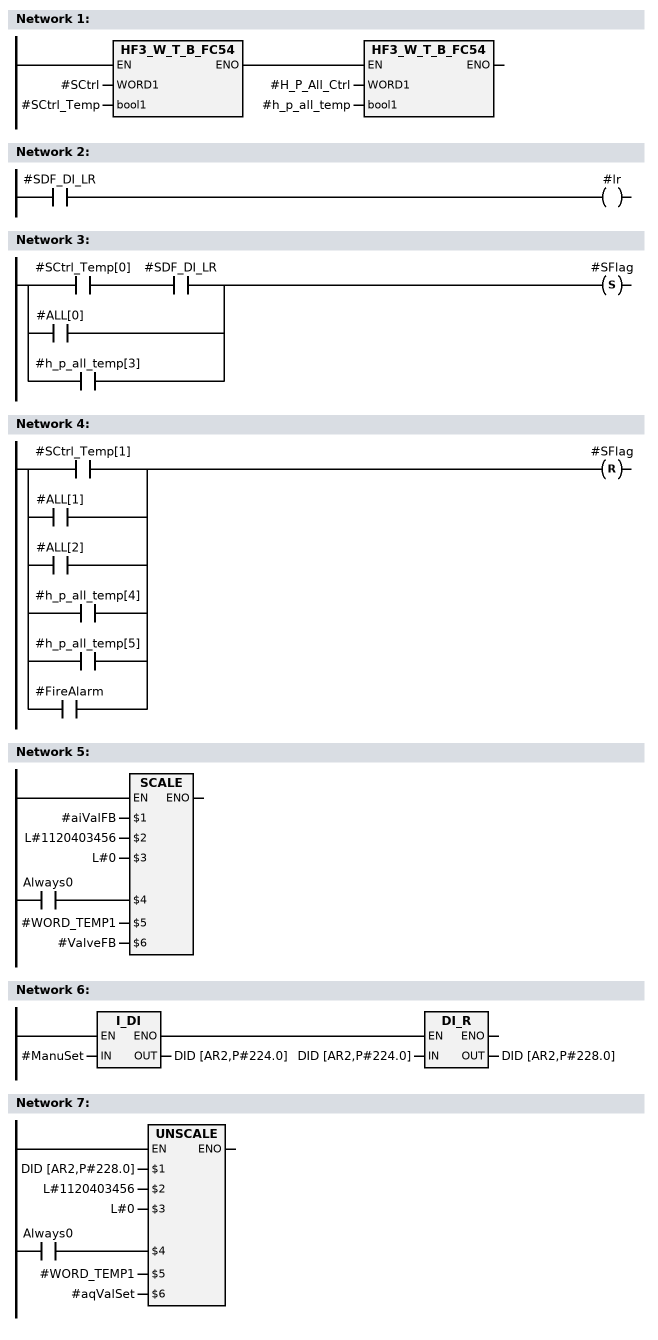
NETWORK
TITLE =
      A(;
      CALL  "HF3_W_T_B_FC54" (
           WORD1                    := #SCtrl,
           bool1                    := #SCtrl_Temp);
      A     BR;
      );
      JNB   _001;
      CALL  "HF3_W_T_B_FC54" (
           WORD1                    := #H_P_All_Ctrl,
           bool1                    := #h_p_all_temp);
_001: NOP   0;
NETWORK
TITLE =
      A     #SDF_DI_LR;
      =     #lr;
NETWORK
TITLE =
      A     #SCtrl_Temp[0];
      A     #SDF_DI_LR;
      O     #ALL[0];
      O     #h_p_all_temp[3];
      S     #SFlag;
NETWORK
TITLE =
      O     #SCtrl_Temp[1];
      O     #ALL[1];
      O     #ALL[2];
      O     #h_p_all_temp[4];
      O     #h_p_all_temp[5];
      O     #FireAlarm;
      R     #SFlag;
NETWORK
TITLE =
      A     "Always0";
      =     L 8.0;
      BLD   103;
      CALL  "SCALE" (
           $1                       := #aiValFB,
           $2                       := L#1120403456,
           $3                       := L#0,
           $4                       := L 8.0,
           $5                       := #WORD_TEMP1,
           $6                       := #ValveFB);
      NOP   0;
NETWORK
TITLE =
      A(;
      L     #ManuSet;
      ITD;
      T     DID [AR2,P#224.0];
      SET;
      SAVE;
      CLR;
      A     BR;
      );
      JNB   _002;
      L     DID [AR2,P#224.0];
      DTR;
      T     DID [AR2,P#228.0];
_002: NOP   0;
NETWORK
TITLE =
      A     "Always0";
      =     L 8.0;
      BLD   103;
      CALL  "UNSCALE" (
           $1                       := DID [AR2,P#228.0],
           $2                       := L#1120403456,
           $3                       := L#0,
           $4                       := L 8.0,
           $5                       := #WORD_TEMP1,
           $6                       := #aqValSet);
      NOP   0;
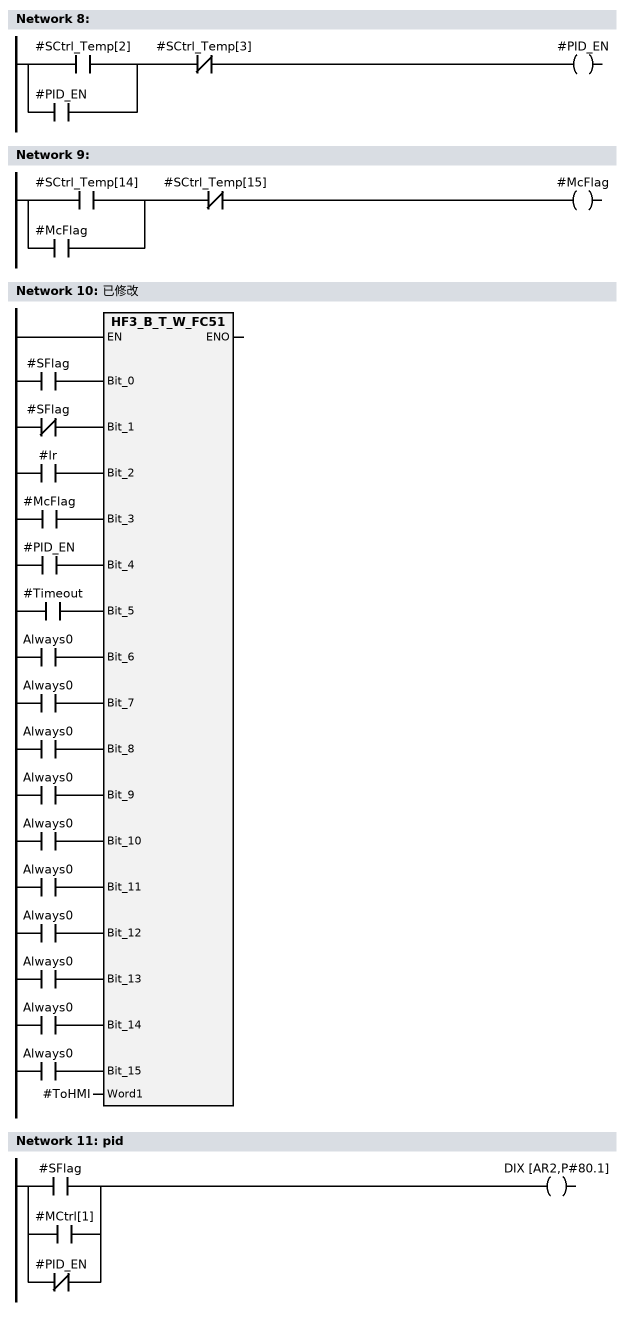
NETWORK
TITLE =
      A(;
      O     #SCtrl_Temp[2];
      O     #PID_EN;
      );
      AN    #SCtrl_Temp[3];
      =     #PID_EN;
NETWORK
TITLE =
      A(;
      O     #SCtrl_Temp[14];
      O     #McFlag;
      );
      AN    #SCtrl_Temp[15];
      =     #McFlag;
NETWORK
TITLE = 已修改
      A     #SFlag;
      =     L 8.0;
      BLD   103;
      AN    #SFlag;
      =     L 8.1;
      BLD   103;
      A     #lr;
      =     L 8.2;
      BLD   103;
      A     #McFlag;
      =     L 8.3;
      BLD   103;
      A     #PID_EN;
      =     L 8.4;
      BLD   103;
      A     #Timeout;
      =     L 8.5;
      BLD   103;
      A     "Always0";
      =     L 8.6;
      BLD   103;
      A     "Always0";
      =     L 8.7;
      BLD   103;
      A     "Always0";
      =     L 9.0;
      BLD   103;
      A     "Always0";
      =     L 9.1;
      BLD   103;
      A     "Always0";
      =     L 9.2;
      BLD   103;
      A     "Always0";
      =     L 9.3;
      BLD   103;
      A     "Always0";
      =     L 9.4;
      BLD   103;
      A     "Always0";
      =     L 9.5;
      BLD   103;
      A     "Always0";
      =     L 9.6;
      BLD   103;
      A     "Always0";
      =     L 9.7;
      BLD   103;
      CALL  "HF3_B_T_W_FC51" (
           Bit_0                    := L 8.0,
           Bit_1                    := L 8.1,
           Bit_2                    := L 8.2,
           Bit_3                    := L 8.3,
           Bit_4                    := L 8.4,
           Bit_5                    := L 8.5,
           Bit_6                    := L 8.6,
           Bit_7                    := L 8.7,
           Bit_8                    := L 9.0,
           Bit_9                    := L 9.1,
           Bit_10                   := L 9.2,
           Bit_11                   := L 9.3,
           Bit_12                   := L 9.4,
           Bit_13                   := L 9.5,
           Bit_14                   := L 9.6,
           Bit_15                   := L 9.7,
           Word1                    := #ToHMI);
      NOP   0;
NETWORK
TITLE = pid
      O     #SFlag;
      O     #MCtrl[1];
      ON    #PID_EN;
      =     DIX [AR2,P#80.1];
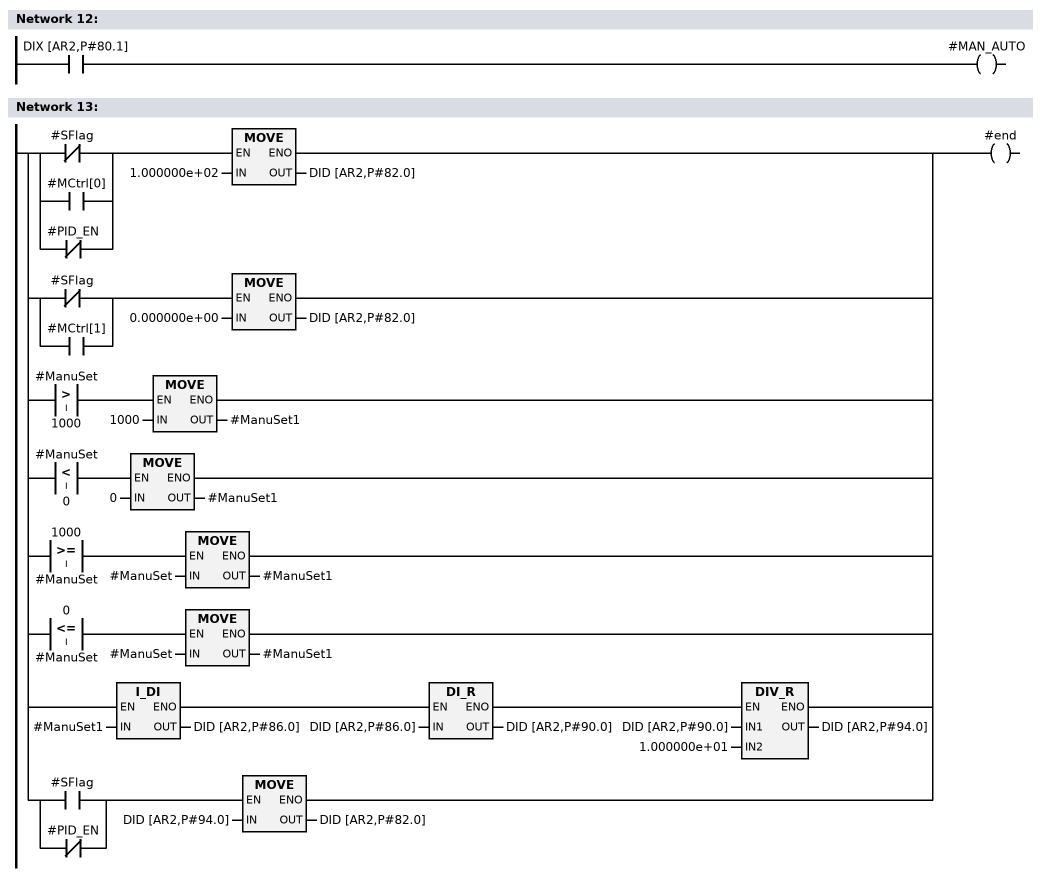
NETWORK
TITLE =
      A     DIX [AR2,P#80.1];
      =     #MAN_AUTO;
NETWORK
TITLE =
      O(;
      A(;
      ON    #SFlag;
      O     #MCtrl[0];
      ON    #PID_EN;
      );
      JNB   _003;
      L     1.000000e+02;
      T     DID [AR2,P#82.0];
      SET;
      SAVE;
      CLR;
_003: A     BR;
      );
      O(;
      A(;
      ON    #SFlag;
      O     #MCtrl[1];
      );
      JNB   _004;
      L     0.000000e+00;
      T     DID [AR2,P#82.0];
      SET;
      SAVE;
      CLR;
_004: A     BR;
      );
      O(;
      A(;
      L     #ManuSet;
      L     1000;
      >I;
      );
      JNB   _005;
      L     1000;
      T     #ManuSet1;
      SET;
      SAVE;
      CLR;
_005: A     BR;
      );
      O(;
      A(;
      L     #ManuSet;
      L     0;
      <I;
      );
      JNB   _006;
      L     0;
      T     #ManuSet1;
      SET;
      SAVE;
      CLR;
_006: A     BR;
      );
      O(;
      A(;
      L     1000;
      L     #ManuSet;
      >=I;
      );
      JNB   _007;
      L     #ManuSet;
      T     #ManuSet1;
      SET;
      SAVE;
      CLR;
_007: A     BR;
      );
      O(;
      A(;
      L     0;
      L     #ManuSet;
      <=I;
      );
      JNB   _008;
      L     #ManuSet;
      T     #ManuSet1;
      SET;
      SAVE;
      CLR;
_008: A     BR;
      );
      O(;
      A(;
      A(;
      L     #ManuSet1;
      ITD;
      T     DID [AR2,P#86.0];
      SET;
      SAVE;
      CLR;
      A     BR;
      );
      JNB   _009;
      L     DID [AR2,P#86.0];
      DTR;
      T     DID [AR2,P#90.0];
      SET;
      SAVE;
      CLR;
_009: A     BR;
      );
      JNB   _00a;
      L     DID [AR2,P#90.0];
      L     1.000000e+01;
      /R;
      T     DID [AR2,P#94.0];
      AN    OV;
      SAVE;
      CLR;
_00a: A     BR;
      );
      O(;
      A(;
      O     #SFlag;
      ON    #PID_EN;
      );
      JNB   _00b;
      L     DID [AR2,P#94.0];
      T     DID [AR2,P#82.0];
      SET;
      SAVE;
      CLR;
_00b: A     BR;
      );
      =     #end;
NETWORK
TITLE =
      A     #MAN_AUTO;
      =     L 8.1;
      BLD   103;
      BLD   14;
      =     L 15.0;
      L     DINO;
      T     LW 13;
      CDB;
      OPN   DI [LW 13];
      TAR2  LD 9;
      A     L 8.1;
      =     DIX [AR2,P#98.1];
      L     L#200;
      T     DID [AR2,P#100.0];
      L     L#1056964608;
      T     DID [AR2,P#134.0];
      +AR2  P#98.0;
      UC    "pid";
      LAR2  LD 9;
      CDB;
      BLD   15;
      NOP   0;
NETWORK
TITLE =
END_FUNCTION_BLOCK

FUNCTION_BLOCK "HF3_FJ_FB2761"	// FB 2761
VERSION : 0.1
VAR
  FJ1 : FB 2762;
END_VAR
BEGIN
NETWORK
TITLE = 高架站风机
      A     M 30.0;
      =     L 0.0;
      BLD   103;
      A     M 30.1;
      =     L 0.1;
      BLD   103;
      A     M 30.2;
      =     L 0.2;
      BLD   103;
      A     M 30.3;
      =     L 0.3;
      BLD   103;
      A     M 30.4;
      =     L 0.4;
      BLD   103;
      A     M 30.5;
      =     L 0.5;
      BLD   103;
      A     M 30.6;
      =     L 0.6;
      BLD   103;
      BLD   14;
      =     L 7.0;
      L     DINO;
      T     LW 5;
      CDB;
      OPN   DI [LW 5];
      TAR2  LD 1;
      L     MW 20;
      T     #FJ1.SCtrl;
      A     L 0.0;
      =     #FJ1.DI_LR;
      A     L 0.1;
      =     #FJ1.DI_Run;
      A     L 0.2;
      =     #FJ1.DI_Stp;
      A     L 0.3;
      =     #FJ1.DI_Flt;
      A     L 0.4;
      =     #FJ1.Stop;
      A     L 0.5;
      =     #FJ1.FireAlarm;
      A     L 0.6;
      =     #FJ1.BlockAlarm;
      L     L#20000;
      T     #FJ1.PT1;
      +AR2  P#0.0;
      UC    "HF3_FJ_FB2762";
      LAR2  LD 1;
      A     #FJ1.DO_Run;
      =     M 40.0;
      A     #FJ1.DO_Stp;
      =     M 40.1;
      CDB;
      BLD   15;
      NOP   0;
END_FUNCTION_BLOCK

FUNCTION_BLOCK "HF3_FJ_FB2762"	// FB 2762
VERSION : 0.1
VAR_INPUT
  SCtrl : WORD ;	//控制命令
  H_P_ALL_Ctrl : WORD ;	//全局命令
  DI_LR : BOOL ;	//远程/就地
  DI_Run : BOOL ;	//运行反馈
  DI_Stp : BOOL ;	//停止反馈
  DI_Flt : BOOL ;	//故障反馈
  Stop : BOOL ;	//连锁信号
  FireAlarm : BOOL ;	//火灾信号
  BlockAlarm : BOOL ;	//阻塞信号
  MCtrl : ARRAY  [0 .. 3 ] OF //模式控制
  BOOL ;
  Mode : ARRAY  [0 .. 15 ] OF //模式执行状态
  BOOL ;
  ALL : ARRAY  [0 .. 15 ] OF //单系统命令
  BOOL ;
  PT1 : TIME ;	//设备动作超时
END_VAR
VAR_OUTPUT
  DO_Run : BOOL ;	//运行控制
  DO_Stp : BOOL ;	//关机控制
  ToHMI : WORD ;	//给上位信号
  RT : INT ;	//运行时间
  SumFlt : INT ;	//故障次数
  SumRun : INT ;	//启动次数
END_VAR
VAR
  SCtrl_Temp : ARRAY  [0 .. 15 ] OF BOOL ;
  DI_Temp : ARRAY  [0 .. 15 ] OF BOOL ;
  DO_Temp : ARRAY  [0 .. 15 ] OF BOOL ;
  H_P_ALL_Ctrl_Temp : ARRAY  [0 .. 15 ] OF BOOL ;
  Ctrl : ARRAY  [0 .. 15 ] OF BOOL ;
  TON1 : SFB 4;
  SFlag : BOOL ;
  QTout : BOOL ;
  Timeout : BOOL ;	//设备动作超时
  Refuse : BOOL ;	//模式不符
  McFlag : BOOL ;	//检修牌
END_VAR
BEGIN
NETWORK
TITLE =
      A(;
      CALL  "HF3_W_T_B_FC54" (
           WORD1                    := #SCtrl,
           bool1                    := #SCtrl_Temp);
      A     BR;
      );
      JNB   _001;
      CALL  "HF3_W_T_B_FC54" (
           WORD1                    := #H_P_ALL_Ctrl,
           bool1                    := #H_P_ALL_Ctrl_Temp);
_001: NOP   0;
NETWORK
TITLE =
      A     #DI_LR;
      =     #DI_Temp[0];
NETWORK
TITLE =
      A     #DI_Run;
      =     #DI_Temp[1];
NETWORK
TITLE =
      A     #DI_Stp;
      =     #DI_Temp[2];
NETWORK
TITLE =
      A     #DI_Flt;
      =     #DI_Temp[3];
NETWORK
TITLE = 单控标志
      O     #SCtrl_Temp[0];
      O     #SCtrl_Temp[0];
      O     #SCtrl_Temp[0];
      S     DIX [AR2,P#58.0];
NETWORK
TITLE = 模控标志
      O     #SCtrl_Temp[1];
      O     #ALL[1];
      O     #H_P_ALL_Ctrl_Temp[4];
      O     #H_P_ALL_Ctrl_Temp[5];
      R     DIX [AR2,P#58.0];
NETWORK
TITLE = 单/模控开
      A     DIX [AR2,P#58.0];
      A     #SCtrl_Temp[2];
      O;
      AN    DIX [AR2,P#58.0];
      A     #MCtrl[0];
      =     #Ctrl[0];
NETWORK
TITLE = 单/模控关
      A     DIX [AR2,P#58.0];
      A     #SCtrl_Temp[3];
      O;
      AN    DIX [AR2,P#58.0];
      A     #MCtrl[1];
      =     #Ctrl[1];
NETWORK
TITLE = 模式预期与实际状态比较
      A     #MCtrl[0];
      AN    #DI_Temp[1];
      O;
      A     #MCtrl[1];
      AN    #DI_Temp[2];
      =     DIX [AR2,P#58.3];
NETWORK
TITLE = 挂牌
      A     #SCtrl_Temp[14];
      AN    #SCtrl_Temp[15];
      S     DIX [AR2,P#58.4];
NETWORK
TITLE = 摘牌
      A     #SCtrl_Temp[15];
      AN    #SCtrl_Temp[14];
      R     DIX [AR2,P#58.4];
NETWORK
TITLE =
      A(;
      O     #Ctrl[14];
      O     #Ctrl[15];
      );
      =     L 0.0;
      BLD   103;
      BLD   16;
      =     L 8.0;
      L     DINO;
      T     LW 6;
      CDB;
      OPN   DI [LW 6];
      TAR2  LD 2;
      A     L 0.0;
      =     DIX [AR2,P#36.0];
      L     L#5000;
      T     DID [AR2,P#38.0];
      +AR2  P#36.0;
      UC    "TON";
      LAR2  LD 2;
      A     DIX [AR2,P#42.0];
      =     DBX [AR2,P#58.1];
      CDB;
      BLD   17;
      NOP   0;
NETWORK
TITLE =
      A     DIX [AR2,P#58.1];
      S     DIX [AR2,P#58.2];
NETWORK
TITLE =
      A     DIX [AR2,P#58.0];
      A(;
      O     #SCtrl_Temp[1];
      O     #SCtrl_Temp[2];
      );
      O;
      AN    DIX [AR2,P#58.0];
      A     #Mode[0];
      O     #SCtrl_Temp[5];
      O     #H_P_ALL_Ctrl_Temp[0];
      R     DIX [AR2,P#58.2];
NETWORK
TITLE =
      A(;
      O     #Ctrl[0];
      O     #DO_Run;
      );
      AN    #Ctrl[1];
      A     #DI_LR;
      AN    #DI_Run;
      AN    #DO_Stp;
      AN    #DI_Flt;
      AN    DIX [AR2,P#58.2];
      =     #DO_Run;
      =     #Ctrl[14];
NETWORK
TITLE =
      A(;
      O     #Ctrl[1];
      O     #DO_Stp;
      );
      AN    #Ctrl[0];
      A     #DI_LR;
      AN    #DI_Stp;
      AN    #DO_Run;
      AN    #DI_Flt;
      AN    DIX [AR2,P#58.2];
      =     #DO_Stp;
      =     #Ctrl[15];
NETWORK
TITLE =
      A     DIX [AR2,P#58.0];
      =     L 0.0;
      BLD   103;
      AN    DIX [AR2,P#58.0];
      =     L 0.1;
      BLD   103;
      A     #DI_LR;
      =     L 0.2;
      BLD   103;
      A     #DI_Run;
      =     L 0.3;
      BLD   103;
      A     #DI_Stp;
      =     L 0.4;
      BLD   103;
      A     #DI_Flt;
      =     L 0.5;
      BLD   103;
      A     DIX [AR2,P#58.3];
      =     L 0.6;
      BLD   103;
      A     DIX [AR2,P#58.2];
      =     L 0.7;
      BLD   103;
      A     DIX [AR2,P#58.4];
      =     L 1.0;
      BLD   103;
      A     "Always0";
      =     L 1.1;
      BLD   103;
      A     "Always0";
      =     L 1.2;
      BLD   103;
      A     "Always0";
      =     L 1.3;
      BLD   103;
      A     "Always0";
      =     L 1.4;
      BLD   103;
      A     "Always0";
      =     L 1.5;
      BLD   103;
      A     "Always0";
      =     L 1.6;
      BLD   103;
      A     "Always0";
      =     L 1.7;
      BLD   103;
      CALL  "HF3_B_T_W_FC51" (
           Bit_0                    := L 0.0,
           Bit_1                    := L 0.1,
           Bit_2                    := L 0.2,
           Bit_3                    := L 0.3,
           Bit_4                    := L 0.4,
           Bit_5                    := L 0.5,
           Bit_6                    := L 0.6,
           Bit_7                    := L 0.7,
           Bit_8                    := L 1.0,
           Bit_9                    := L 1.1,
           Bit_10                   := L 1.2,
           Bit_11                   := L 1.3,
           Bit_12                   := L 1.4,
           Bit_13                   := L 1.5,
           Bit_14                   := L 1.6,
           Bit_15                   := L 1.7,
           Word1                    := #ToHMI);
      NOP   0;
NETWORK
TITLE =
END_FUNCTION_BLOCK

